    |   movel([0.066867, -1.321516, -2.613726, -0.777146, 1.570796, 1.637663],accel_mss,speed_ms,0,blend_radius_m)
    |   movel([0.067167, -1.321241, -2.613897, -0.777250, 1.570796, 1.637963],accel_mss,speed_ms,0,blend_radius_m)
    |   movel([0.067720, -1.320799, -2.614173, -0.777418, 1.570796, 1.638516],accel_mss,speed_ms,0,blend_radius_m)
    |   movel([0.068900, -1.319924, -2.614716, -0.777749, 1.570796, 1.639696],accel_mss,speed_ms,0,blend_radius_m)
    |   movel([0.070231, -1.318957, -2.615316, -0.778116, 1.570796, 1.641027],accel_mss,speed_ms,0,blend_radius_m)
    |   movel([0.071504, -1.318055, -2.615874, -0.778460, 1.570796, 1.642300],accel_mss,speed_ms,0,blend_radius_m)
    |   movel([0.073287, -1.316906, -2.616583, -0.778900, 1.570796, 1.644084],accel_mss,speed_ms,0,blend_radius_m)
    |   movel([0.076248, -1.315195, -2.617636, -0.779558, 1.570796, 1.647044],accel_mss,speed_ms,0,blend_radius_m)
    |   movel([0.079336, -1.313494, -2.618679, -0.780215, 1.570796, 1.650133],accel_mss,speed_ms,0,blend_radius_m)
    |   movel([0.081717, -1.312291, -2.619415, -0.780683, 1.570796, 1.652514],accel_mss,speed_ms,0,blend_radius_m)
    |   movel([0.083889, -1.311300, -2.620019, -0.781070, 1.570796, 1.654686],accel_mss,speed_ms,0,blend_radius_m)
    |   movel([0.085940, -1.310444, -2.620540, -0.781405, 1.570796, 1.656736],accel_mss,speed_ms,0,blend_radius_m)
    |   movel([0.088113, -1.309632, -2.621034, -0.781723, 1.570796, 1.658909],accel_mss,speed_ms,0,blend_radius_m)
    |   movel([0.090652, -1.308770, -2.621556, -0.782062, 1.570796, 1.661449],accel_mss,speed_ms,0,blend_radius_m)
    |   movel([0.093223, -1.307968, -2.622042, -0.782379, 1.570796, 1.664019],accel_mss,speed_ms,0,blend_radius_m)
    |   movel([0.095145, -1.307454, -2.622353, -0.782582, 1.570796, 1.665941],accel_mss,speed_ms,0,blend_radius_m)
    |   movel([0.096536, -1.307182, -2.622517, -0.782690, 1.570796, 1.667333],accel_mss,speed_ms,0,blend_radius_m)
    |   movel([0.097274, -1.307208, -2.622501, -0.782680, 1.570796, 1.668070],accel_mss,speed_ms,0,blend_radius_m)
    |   movel([0.097500, -1.307382, -2.622396, -0.782611, 1.570796, 1.668297],accel_mss,speed_ms,0,blend_radius_m)
    |   movel([0.097411, -1.307944, -2.622056, -0.782389, 1.570796, 1.668208],accel_mss,speed_ms,0,blend_radius_m)
    |   movel([0.097336, -1.308222, -2.621888, -0.782279, 1.570796, 1.668132],accel_mss,speed_ms,0,blend_radius_m)
    |   movel([0.097240, -1.308511, -2.621713, -0.782165, 1.570796, 1.668037],accel_mss,speed_ms,0,blend_radius_m)
    |   movel([0.097140, -1.308774, -2.621554, -0.782061, 1.570796, 1.667936],accel_mss,speed_ms,0,blend_radius_m)
    |   speed_ms = 0.003
    |   movel([0.097054, -1.295189, -2.614952, -0.802248, 1.570796, 1.667851],accel_mss,speed_ms,0,blend_radius_m)
    |   speed_ms = 1.000
    |   movel([0.097054, -1.268961, -2.601575, -0.841853, 1.570796, 1.667851],accel_mss,speed_ms,0,blend_radius_m)
    |   movel([0.095455, -1.266877, -2.602766, -0.842746, 1.570796, 1.666251],accel_mss,speed_ms,0,blend_radius_m)
    |   movel([0.095455, -1.293135, -2.616170, -0.803084, 1.570796, 1.666251],accel_mss,speed_ms,0,blend_radius_m)
    |   speed_ms = 0.003
    |   movel([0.095455, -1.303429, -2.621063, -0.787897, 1.570796, 1.666251],accel_mss,speed_ms,0,blend_radius_m)
    |   speed_ms = 0.007
    |   movel([0.094815, -1.303693, -2.620905, -0.787791, 1.570796, 1.665611],accel_mss,speed_ms,0,blend_radius_m)
    |   movel([0.093768, -1.303954, -2.620748, -0.787687, 1.570796, 1.664565],accel_mss,speed_ms,0,blend_radius_m)
    |   movel([0.093133, -1.304102, -2.620659, -0.787628, 1.570796, 1.663930],accel_mss,speed_ms,0,blend_radius_m)
    |   movel([0.092577, -1.304211, -2.620593, -0.787584, 1.570796, 1.663373],accel_mss,speed_ms,0,blend_radius_m)
    |   movel([0.092119, -1.304286, -2.620548, -0.787555, 1.570796, 1.662915],accel_mss,speed_ms,0,blend_radius_m)
    |   movel([0.091857, -1.304106, -2.620657, -0.787627, 1.570796, 1.662654],accel_mss,speed_ms,0,blend_radius_m)
    |   movel([0.091804, -1.303854, -2.620808, -0.787727, 1.570796, 1.662600],accel_mss,speed_ms,0,blend_radius_m)
    |   movel([0.091848, -1.303588, -2.620968, -0.787833, 1.570796, 1.662644],accel_mss,speed_ms,0,blend_radius_m)
    |   movel([0.092415, -1.303110, -2.621254, -0.788024, 1.570796, 1.663211],accel_mss,speed_ms,0,blend_radius_m)
    |   movel([0.093796, -1.302701, -2.621500, -0.788188, 1.570796, 1.664592],accel_mss,speed_ms,0,blend_radius_m)
    |   movel([0.095147, -1.302357, -2.621706, -0.788326, 1.570796, 1.665943],accel_mss,speed_ms,0,blend_radius_m)
    |   movel([0.095680, -1.302353, -2.621709, -0.788328, 1.570796, 1.666476],accel_mss,speed_ms,0,blend_radius_m)
    |   movel([0.095880, -1.302466, -2.621641, -0.788282, 1.570796, 1.666676],accel_mss,speed_ms,0,blend_radius_m)
    |   movel([0.095874, -1.302908, -2.621376, -0.788105, 1.570796, 1.666670],accel_mss,speed_ms,0,blend_radius_m)
    |   movel([0.095665, -1.303223, -2.621187, -0.787979, 1.570796, 1.666461],accel_mss,speed_ms,0,blend_radius_m)
    |   speed_ms = 0.003
    |   movel([0.095455, -1.306916, -2.622678, -0.782796, 1.570796, 1.666251],accel_mss,speed_ms,0,blend_radius_m)
    |   speed_ms = 0.007
    |   movel([0.094815, -1.307179, -2.622519, -0.782691, 1.570796, 1.665611],accel_mss,speed_ms,0,blend_radius_m)
    |   movel([0.093768, -1.307439, -2.622362, -0.782588, 1.570796, 1.664565],accel_mss,speed_ms,0,blend_radius_m)
    |   movel([0.093133, -1.307587, -2.622272, -0.782530, 1.570796, 1.663930],accel_mss,speed_ms,0,blend_radius_m)
    |   movel([0.092577, -1.307696, -2.622206, -0.782487, 1.570796, 1.663373],accel_mss,speed_ms,0,blend_radius_m)
    |   movel([0.092119, -1.307771, -2.622161, -0.782457, 1.570796, 1.662915],accel_mss,speed_ms,0,blend_radius_m)
    |   movel([0.091857, -1.307590, -2.622270, -0.782528, 1.570796, 1.662654],accel_mss,speed_ms,0,blend_radius_m)
    |   movel([0.091804, -1.307340, -2.622422, -0.782628, 1.570796, 1.662600],accel_mss,speed_ms,0,blend_radius_m)
    |   movel([0.091848, -1.307074, -2.622582, -0.782733, 1.570796, 1.662644],accel_mss,speed_ms,0,blend_radius_m)
    |   movel([0.092415, -1.306598, -2.622870, -0.782922, 1.570796, 1.663211],accel_mss,speed_ms,0,blend_radius_m)
    |   movel([0.093796, -1.306189, -2.623116, -0.783084, 1.570796, 1.664592],accel_mss,speed_ms,0,blend_radius_m)
    |   movel([0.095147, -1.305846, -2.623322, -0.783220, 1.570796, 1.665943],accel_mss,speed_ms,0,blend_radius_m)
    |   movel([0.095680, -1.305842, -2.623325, -0.783222, 1.570796, 1.666476],accel_mss,speed_ms,0,blend_radius_m)
    |   movel([0.095880, -1.305954, -2.623257, -0.783177, 1.570796, 1.666676],accel_mss,speed_ms,0,blend_radius_m)
    |   movel([0.095874, -1.306395, -2.622992, -0.783002, 1.570796, 1.666670],accel_mss,speed_ms,0,blend_radius_m)
    |   movel([0.095665, -1.306710, -2.622802, -0.782877, 1.570796, 1.666461],accel_mss,speed_ms,0,blend_radius_m)
    |   speed_ms = 0.003
    |   movel([0.095455, -1.293135, -2.616170, -0.803084, 1.570796, 1.666251],accel_mss,speed_ms,0,blend_radius_m)
    |   speed_ms = 1.000
    |   movel([0.095455, -1.266877, -2.602766, -0.842746, 1.570796, 1.666251],accel_mss,speed_ms,0,blend_radius_m)
    |   movel([0.095405, -1.265298, -2.603664, -0.843426, 1.570796, 1.666201],accel_mss,speed_ms,0,blend_radius_m)
    |   movel([0.095405, -1.291578, -2.617089, -0.803722, 1.570796, 1.666201],accel_mss,speed_ms,0,blend_radius_m)
    |   speed_ms = 0.003
    |   movel([0.095405, -1.301882, -2.621990, -0.788516, 1.570796, 1.666201],accel_mss,speed_ms,0,blend_radius_m)
    |   speed_ms = 0.007
    |   movel([0.093973, -1.302304, -2.621738, -0.788347, 1.570796, 1.664770],accel_mss,speed_ms,0,blend_radius_m)
    |   movel([0.092537, -1.302698, -2.621502, -0.788189, 1.570796, 1.663334],accel_mss,speed_ms,0,blend_radius_m)
    |   movel([0.092269, -1.302658, -2.621526, -0.788205, 1.570796, 1.663065],accel_mss,speed_ms,0,blend_radius_m)
    |   movel([0.092184, -1.302449, -2.621651, -0.788289, 1.570796, 1.662981],accel_mss,speed_ms,0,blend_radius_m)
    |   movel([0.092128, -1.302079, -2.621873, -0.788437, 1.570796, 1.662924],accel_mss,speed_ms,0,blend_radius_m)
    |   movel([0.092124, -1.301814, -2.622031, -0.788544, 1.570796, 1.662920],accel_mss,speed_ms,0,blend_radius_m)
    |   movel([0.092244, -1.301453, -2.622247, -0.788689, 1.570796, 1.663040],accel_mss,speed_ms,0,blend_radius_m)
    |   movel([0.093053, -1.300803, -2.622635, -0.788951, 1.570796, 1.663849],accel_mss,speed_ms,0,blend_radius_m)
    |   movel([0.094199, -1.300463, -2.622838, -0.789088, 1.570796, 1.664996],accel_mss,speed_ms,0,blend_radius_m)
    |   movel([0.095309, -1.300319, -2.622924, -0.789146, 1.570796, 1.666105],accel_mss,speed_ms,0,blend_radius_m)
    |   movel([0.095864, -1.300514, -2.622808, -0.789067, 1.570796, 1.666660],accel_mss,speed_ms,0,blend_radius_m)
    |   movel([0.095977, -1.300744, -2.622670, -0.788974, 1.570796, 1.666773],accel_mss,speed_ms,0,blend_radius_m)
    |   movel([0.095993, -1.301082, -2.622469, -0.788838, 1.570796, 1.666789],accel_mss,speed_ms,0,blend_radius_m)
    |   movel([0.095919, -1.301425, -2.622264, -0.788700, 1.570796, 1.666715],accel_mss,speed_ms,0,blend_radius_m)
    |   movel([0.095405, -1.301882, -2.621990, -0.788516, 1.570796, 1.666201],accel_mss,speed_ms,0,blend_radius_m)
    |   speed_ms = 0.003
    |   movel([0.095405, -1.305372, -2.623608, -0.783409, 1.570796, 1.666201],accel_mss,speed_ms,0,blend_radius_m)
    |   speed_ms = 0.007
    |   movel([0.093973, -1.305793, -2.623354, -0.783242, 1.570796, 1.664770],accel_mss,speed_ms,0,blend_radius_m)
    |   movel([0.092537, -1.306187, -2.623117, -0.783085, 1.570796, 1.663334],accel_mss,speed_ms,0,blend_radius_m)
    |   movel([0.092269, -1.306146, -2.623142, -0.783101, 1.570796, 1.663065],accel_mss,speed_ms,0,blend_radius_m)
    |   movel([0.092184, -1.305938, -2.623267, -0.783184, 1.570796, 1.662981],accel_mss,speed_ms,0,blend_radius_m)
    |   movel([0.092128, -1.305569, -2.623489, -0.783331, 1.570796, 1.662924],accel_mss,speed_ms,0,blend_radius_m)
    |   movel([0.092124, -1.305304, -2.623649, -0.783437, 1.570796, 1.662920],accel_mss,speed_ms,0,blend_radius_m)
    |   movel([0.092244, -1.304944, -2.623865, -0.783580, 1.570796, 1.663040],accel_mss,speed_ms,0,blend_radius_m)
    |   movel([0.093053, -1.304296, -2.624254, -0.783839, 1.570796, 1.663849],accel_mss,speed_ms,0,blend_radius_m)
    |   movel([0.094199, -1.303956, -2.624458, -0.783975, 1.570796, 1.664996],accel_mss,speed_ms,0,blend_radius_m)
    |   movel([0.095309, -1.303812, -2.624544, -0.784033, 1.570796, 1.666105],accel_mss,speed_ms,0,blend_radius_m)
    |   movel([0.095864, -1.304007, -2.624428, -0.783955, 1.570796, 1.666660],accel_mss,speed_ms,0,blend_radius_m)
    |   movel([0.095977, -1.304237, -2.624289, -0.783863, 1.570796, 1.666773],accel_mss,speed_ms,0,blend_radius_m)
    |   movel([0.095993, -1.304573, -2.624088, -0.783728, 1.570796, 1.666789],accel_mss,speed_ms,0,blend_radius_m)
    |   movel([0.095919, -1.304916, -2.623882, -0.783591, 1.570796, 1.666715],accel_mss,speed_ms,0,blend_radius_m)
    |   movel([0.095405, -1.305372, -2.623608, -0.783409, 1.570796, 1.666201],accel_mss,speed_ms,0,blend_radius_m)
    |   speed_ms = 0.003
    |   movel([0.095405, -1.291578, -2.617089, -0.803722, 1.570796, 1.666201],accel_mss,speed_ms,0,blend_radius_m)
    |   speed_ms = 1.000
    |   movel([0.095405, -1.265298, -2.603664, -0.843426, 1.570796, 1.666201],accel_mss,speed_ms,0,blend_radius_m)
    |   movel([0.086620, -1.269064, -2.601516, -0.841809, 1.570796, 1.657416],accel_mss,speed_ms,0,blend_radius_m)
    |   movel([0.086620, -1.295291, -2.614891, -0.802207, 1.570796, 1.657416],accel_mss,speed_ms,0,blend_radius_m)
    |   speed_ms = 0.003
    |   movel([0.086620, -1.305571, -2.619774, -0.787044, 1.570796, 1.657416],accel_mss,speed_ms,0,blend_radius_m)
    |   speed_ms = 0.007
    |   movel([0.086582, -1.306010, -2.619509, -0.786870, 1.570796, 1.657378],accel_mss,speed_ms,0,blend_radius_m)
    |   movel([0.086379, -1.306296, -2.619337, -0.786757, 1.570796, 1.657175],accel_mss,speed_ms,0,blend_radius_m)
    |   movel([0.085833, -1.306567, -2.619173, -0.786649, 1.570796, 1.656630],accel_mss,speed_ms,0,blend_radius_m)
    |   movel([0.085166, -1.306876, -2.618986, -0.786527, 1.570796, 1.655962],accel_mss,speed_ms,0,blend_radius_m)
    |   movel([0.084376, -1.307221, -2.618777, -0.786391, 1.570796, 1.655172],accel_mss,speed_ms,0,blend_radius_m)
    |   movel([0.082276, -1.308128, -2.618228, -0.786033, 1.570796, 1.653073],accel_mss,speed_ms,0,blend_radius_m)
    |   movel([0.080804, -1.308806, -2.617816, -0.785767, 1.570796, 1.651600],accel_mss,speed_ms,0,blend_radius_m)
    |   movel([0.079595, -1.309416, -2.617445, -0.785528, 1.570796, 1.650391],accel_mss,speed_ms,0,blend_radius_m)
    |   movel([0.078387, -1.310089, -2.617036, -0.785264, 1.570796, 1.649183],accel_mss,speed_ms,0,blend_radius_m)
    |   movel([0.077797, -1.310425, -2.616831, -0.785133, 1.570796, 1.648593],accel_mss,speed_ms,0,blend_radius_m)
    |   movel([0.077272, -1.310708, -2.616659, -0.785023, 1.570796, 1.648069],accel_mss,speed_ms,0,blend_radius_m)
    |   movel([0.076832, -1.310931, -2.616522, -0.784935, 1.570796, 1.647629],accel_mss,speed_ms,0,blend_radius_m)
    |   movel([0.076556, -1.310865, -2.616563, -0.784961, 1.570796, 1.647352],accel_mss,speed_ms,0,blend_radius_m)
    |   movel([0.076460, -1.310625, -2.616709, -0.785055, 1.570796, 1.647257],accel_mss,speed_ms,0,blend_radius_m)
    |   movel([0.076484, -1.310298, -2.616908, -0.785183, 1.570796, 1.647280],accel_mss,speed_ms,0,blend_radius_m)
    |   movel([0.076654, -1.309989, -2.617097, -0.785303, 1.570796, 1.647450],accel_mss,speed_ms,0,blend_radius_m)
    |   movel([0.077020, -1.309644, -2.617307, -0.785438, 1.570796, 1.647816],accel_mss,speed_ms,0,blend_radius_m)
    |   movel([0.077663, -1.309194, -2.617580, -0.785615, 1.570796, 1.648459],accel_mss,speed_ms,0,blend_radius_m)
    |   movel([0.078607, -1.308648, -2.617912, -0.785829, 1.570796, 1.649403],accel_mss,speed_ms,0,blend_radius_m)
    |   movel([0.080873, -1.307513, -2.618601, -0.786276, 1.570796, 1.651669],accel_mss,speed_ms,0,blend_radius_m)
    |   movel([0.083162, -1.306405, -2.619271, -0.786713, 1.570796, 1.653958],accel_mss,speed_ms,0,blend_radius_m)
    |   movel([0.084650, -1.305747, -2.619668, -0.786974, 1.570796, 1.655447],accel_mss,speed_ms,0,blend_radius_m)
    |   movel([0.085312, -1.305509, -2.619812, -0.787068, 1.570796, 1.656108],accel_mss,speed_ms,0,blend_radius_m)
    |   movel([0.085892, -1.305370, -2.619896, -0.787124, 1.570796, 1.656689],accel_mss,speed_ms,0,blend_radius_m)
    |   movel([0.086338, -1.305334, -2.619917, -0.787138, 1.570796, 1.657135],accel_mss,speed_ms,0,blend_radius_m)
    |   movel([0.086557, -1.305429, -2.619860, -0.787100, 1.570796, 1.657353],accel_mss,speed_ms,0,blend_radius_m)
    |   speed_ms = 0.003
    |   movel([0.086620, -1.309053, -2.621385, -0.781951, 1.570796, 1.657416],accel_mss,speed_ms,0,blend_radius_m)
    |   speed_ms = 0.007
    |   movel([0.086582, -1.309490, -2.621120, -0.781779, 1.570796, 1.657378],accel_mss,speed_ms,0,blend_radius_m)
    |   movel([0.086379, -1.309776, -2.620947, -0.781667, 1.570796, 1.657175],accel_mss,speed_ms,0,blend_radius_m)
    |   movel([0.085833, -1.310046, -2.620782, -0.781561, 1.570796, 1.656630],accel_mss,speed_ms,0,blend_radius_m)
    |   movel([0.085166, -1.310354, -2.620595, -0.781440, 1.570796, 1.655962],accel_mss,speed_ms,0,blend_radius_m)
    |   movel([0.084376, -1.310699, -2.620385, -0.781305, 1.570796, 1.655172],accel_mss,speed_ms,0,blend_radius_m)
    |   movel([0.082276, -1.311603, -2.619834, -0.780951, 1.570796, 1.653073],accel_mss,speed_ms,0,blend_radius_m)
    |   movel([0.080804, -1.312280, -2.619421, -0.780687, 1.570796, 1.651600],accel_mss,speed_ms,0,blend_radius_m)
    |   movel([0.079595, -1.312889, -2.619050, -0.780450, 1.570796, 1.650391],accel_mss,speed_ms,0,blend_radius_m)
    |   movel([0.078387, -1.313560, -2.618639, -0.780190, 1.570796, 1.649183],accel_mss,speed_ms,0,blend_radius_m)
    |   movel([0.077797, -1.313896, -2.618434, -0.780060, 1.570796, 1.648593],accel_mss,speed_ms,0,blend_radius_m)
    |   movel([0.077272, -1.314177, -2.618261, -0.779951, 1.570796, 1.648069],accel_mss,speed_ms,0,blend_radius_m)
    |   movel([0.076832, -1.314401, -2.618124, -0.779864, 1.570796, 1.647629],accel_mss,speed_ms,0,blend_radius_m)
    |   movel([0.076556, -1.314335, -2.618165, -0.779890, 1.570796, 1.647352],accel_mss,speed_ms,0,blend_radius_m)
    |   movel([0.076460, -1.314095, -2.618312, -0.779983, 1.570796, 1.647257],accel_mss,speed_ms,0,blend_radius_m)
    |   movel([0.076484, -1.313769, -2.618511, -0.780109, 1.570796, 1.647280],accel_mss,speed_ms,0,blend_radius_m)
    |   movel([0.076654, -1.313460, -2.618700, -0.780229, 1.570796, 1.647450],accel_mss,speed_ms,0,blend_radius_m)
    |   movel([0.077020, -1.313116, -2.618911, -0.780362, 1.570796, 1.647816],accel_mss,speed_ms,0,blend_radius_m)
    |   movel([0.077663, -1.312667, -2.619185, -0.780537, 1.570796, 1.648459],accel_mss,speed_ms,0,blend_radius_m)
    |   movel([0.078607, -1.312122, -2.619518, -0.780749, 1.570796, 1.649403],accel_mss,speed_ms,0,blend_radius_m)
    |   movel([0.080873, -1.310990, -2.620208, -0.781191, 1.570796, 1.651669],accel_mss,speed_ms,0,blend_radius_m)
    |   movel([0.083162, -1.309885, -2.620880, -0.781624, 1.570796, 1.653958],accel_mss,speed_ms,0,blend_radius_m)
    |   movel([0.084650, -1.309228, -2.621279, -0.781882, 1.570796, 1.655447],accel_mss,speed_ms,0,blend_radius_m)
    |   movel([0.085312, -1.308990, -2.621423, -0.781976, 1.570796, 1.656108],accel_mss,speed_ms,0,blend_radius_m)
    |   movel([0.085892, -1.308852, -2.621507, -0.782030, 1.570796, 1.656689],accel_mss,speed_ms,0,blend_radius_m)
    |   movel([0.086338, -1.308816, -2.621529, -0.782044, 1.570796, 1.657135],accel_mss,speed_ms,0,blend_radius_m)
    |   movel([0.086557, -1.308911, -2.621471, -0.782007, 1.570796, 1.657353],accel_mss,speed_ms,0,blend_radius_m)
    |   speed_ms = 0.003
    |   movel([0.086620, -1.295291, -2.614891, -0.802207, 1.570796, 1.657416],accel_mss,speed_ms,0,blend_radius_m)
    |   speed_ms = 1.000
    |   movel([0.086620, -1.269064, -2.601516, -0.841809, 1.570796, 1.657416],accel_mss,speed_ms,0,blend_radius_m)
    |   movel([0.086236, -1.268202, -2.602010, -0.842178, 1.570796, 1.657033],accel_mss,speed_ms,0,blend_radius_m)
    |   movel([0.086236, -1.294441, -2.615396, -0.802552, 1.570796, 1.657033],accel_mss,speed_ms,0,blend_radius_m)
    |   speed_ms = 0.003
    |   movel([0.086236, -1.304727, -2.620283, -0.787379, 1.570796, 1.657033],accel_mss,speed_ms,0,blend_radius_m)
    |   speed_ms = 0.007
    |   movel([0.085836, -1.304918, -2.620168, -0.787303, 1.570796, 1.656632],accel_mss,speed_ms,0,blend_radius_m)
    |   movel([0.085399, -1.305046, -2.620090, -0.787252, 1.570796, 1.656196],accel_mss,speed_ms,0,blend_radius_m)
    |   movel([0.085110, -1.304940, -2.620155, -0.787294, 1.570796, 1.655906],accel_mss,speed_ms,0,blend_radius_m)
    |   movel([0.085056, -1.304704, -2.620297, -0.787388, 1.570796, 1.655852],accel_mss,speed_ms,0,blend_radius_m)
    |   movel([0.085010, -1.304411, -2.620473, -0.787505, 1.570796, 1.655807],accel_mss,speed_ms,0,blend_radius_m)
    |   movel([0.084978, -1.304084, -2.620670, -0.787635, 1.570796, 1.655775],accel_mss,speed_ms,0,blend_radius_m)
    |   movel([0.084892, -1.303468, -2.621040, -0.787881, 1.570796, 1.655688],accel_mss,speed_ms,0,blend_radius_m)
    |   movel([0.084735, -1.303084, -2.621270, -0.788035, 1.570796, 1.655531],accel_mss,speed_ms,0,blend_radius_m)
    |   movel([0.084474, -1.302865, -2.621402, -0.788122, 1.570796, 1.655271],accel_mss,speed_ms,0,blend_radius_m)
    |   movel([0.084085, -1.302763, -2.621463, -0.788163, 1.570796, 1.654882],accel_mss,speed_ms,0,blend_radius_m)
    |   movel([0.083756, -1.302782, -2.621451, -0.788155, 1.570796, 1.654553],accel_mss,speed_ms,0,blend_radius_m)
    |   movel([0.083385, -1.302888, -2.621388, -0.788113, 1.570796, 1.654181],accel_mss,speed_ms,0,blend_radius_m)
    |   movel([0.082789, -1.303141, -2.621236, -0.788012, 1.570796, 1.653585],accel_mss,speed_ms,0,blend_radius_m)
    |   movel([0.081437, -1.303782, -2.620851, -0.787756, 1.570796, 1.652233],accel_mss,speed_ms,0,blend_radius_m)
    |   movel([0.079639, -1.304655, -2.620326, -0.787408, 1.570796, 1.650435],accel_mss,speed_ms,0,blend_radius_m)
    |   movel([0.078834, -1.305092, -2.620063, -0.787234, 1.570796, 1.649630],accel_mss,speed_ms,0,blend_radius_m)
    |   movel([0.078346, -1.305441, -2.619853, -0.787095, 1.570796, 1.649142],accel_mss,speed_ms,0,blend_radius_m)
    |   movel([0.077948, -1.305852, -2.619605, -0.786932, 1.570796, 1.648744],accel_mss,speed_ms,0,blend_radius_m)
    |   movel([0.077690, -1.306269, -2.619353, -0.786767, 1.570796, 1.648486],accel_mss,speed_ms,0,blend_radius_m)
    |   movel([0.077544, -1.306721, -2.619080, -0.786588, 1.570796, 1.648340],accel_mss,speed_ms,0,blend_radius_m)
    |   movel([0.077508, -1.307216, -2.618780, -0.786393, 1.570796, 1.648304],accel_mss,speed_ms,0,blend_radius_m)
    |   movel([0.077587, -1.307758, -2.618452, -0.786179, 1.570796, 1.648383],accel_mss,speed_ms,0,blend_radius_m)
    |   movel([0.077671, -1.308128, -2.618228, -0.786033, 1.570796, 1.648467],accel_mss,speed_ms,0,blend_radius_m)
    |   movel([0.077735, -1.308415, -2.618054, -0.785921, 1.570796, 1.648531],accel_mss,speed_ms,0,blend_radius_m)
    |   movel([0.077659, -1.308677, -2.617895, -0.785818, 1.570796, 1.648455],accel_mss,speed_ms,0,blend_radius_m)
    |   movel([0.077187, -1.309039, -2.617674, -0.785675, 1.570796, 1.647984],accel_mss,speed_ms,0,blend_radius_m)
    |   movel([0.076724, -1.309309, -2.617511, -0.785570, 1.570796, 1.647520],accel_mss,speed_ms,0,blend_radius_m)
    |   movel([0.076338, -1.309187, -2.617585, -0.785618, 1.570796, 1.647134],accel_mss,speed_ms,0,blend_radius_m)
    |   movel([0.076209, -1.308628, -2.617924, -0.785837, 1.570796, 1.647005],accel_mss,speed_ms,0,blend_radius_m)
    |   movel([0.076116, -1.307960, -2.618330, -0.786100, 1.570796, 1.646913],accel_mss,speed_ms,0,blend_radius_m)
    |   movel([0.076083, -1.307280, -2.618742, -0.786368, 1.570796, 1.646879],accel_mss,speed_ms,0,blend_radius_m)
    |   movel([0.076095, -1.306774, -2.619048, -0.786567, 1.570796, 1.646891],accel_mss,speed_ms,0,blend_radius_m)
    |   movel([0.076142, -1.306449, -2.619244, -0.786696, 1.570796, 1.646938],accel_mss,speed_ms,0,blend_radius_m)
    |   movel([0.076248, -1.306149, -2.619426, -0.786815, 1.570796, 1.647044],accel_mss,speed_ms,0,blend_radius_m)
    |   movel([0.076446, -1.305763, -2.619659, -0.786968, 1.570796, 1.647243],accel_mss,speed_ms,0,blend_radius_m)
    |   movel([0.076797, -1.305253, -2.619966, -0.787170, 1.570796, 1.647593],accel_mss,speed_ms,0,blend_radius_m)
    |   movel([0.077222, -1.304834, -2.620218, -0.787337, 1.570796, 1.648018],accel_mss,speed_ms,0,blend_radius_m)
    |   movel([0.077828, -1.304417, -2.620470, -0.787503, 1.570796, 1.648625],accel_mss,speed_ms,0,blend_radius_m)
    |   movel([0.078794, -1.303880, -2.620792, -0.787717, 1.570796, 1.649591],accel_mss,speed_ms,0,blend_radius_m)
    |   movel([0.080203, -1.303163, -2.621223, -0.788003, 1.570796, 1.651000],accel_mss,speed_ms,0,blend_radius_m)
    |   movel([0.081785, -1.302416, -2.621671, -0.788302, 1.570796, 1.652581],accel_mss,speed_ms,0,blend_radius_m)
    |   movel([0.083247, -1.301763, -2.622062, -0.788564, 1.570796, 1.654043],accel_mss,speed_ms,0,blend_radius_m)
    |   movel([0.084162, -1.301411, -2.622272, -0.788706, 1.570796, 1.654958],accel_mss,speed_ms,0,blend_radius_m)
    |   movel([0.084675, -1.301251, -2.622368, -0.788770, 1.570796, 1.655472],accel_mss,speed_ms,0,blend_radius_m)
    |   movel([0.084988, -1.301189, -2.622405, -0.788795, 1.570796, 1.655784],accel_mss,speed_ms,0,blend_radius_m)
    |   movel([0.085477, -1.301278, -2.622352, -0.788759, 1.570796, 1.656273],accel_mss,speed_ms,0,blend_radius_m)
    |   movel([0.085801, -1.301477, -2.622233, -0.788679, 1.570796, 1.656597],accel_mss,speed_ms,0,blend_radius_m)
    |   movel([0.086025, -1.301709, -2.622094, -0.788586, 1.570796, 1.656822],accel_mss,speed_ms,0,blend_radius_m)
    |   movel([0.086213, -1.302208, -2.621795, -0.788386, 1.570796, 1.657010],accel_mss,speed_ms,0,blend_radius_m)
    |   movel([0.086374, -1.303118, -2.621250, -0.788021, 1.570796, 1.657170],accel_mss,speed_ms,0,blend_radius_m)
    |   movel([0.086472, -1.304054, -2.620688, -0.787647, 1.570796, 1.657269],accel_mss,speed_ms,0,blend_radius_m)
    |   movel([0.086421, -1.304572, -2.620376, -0.787441, 1.570796, 1.657218],accel_mss,speed_ms,0,blend_radius_m)
    |   speed_ms = 0.003
    |   movel([0.086236, -1.308210, -2.621895, -0.782283, 1.570796, 1.657033],accel_mss,speed_ms,0,blend_radius_m)
    |   speed_ms = 0.007
    |   movel([0.085836, -1.308401, -2.621780, -0.782208, 1.570796, 1.656632],accel_mss,speed_ms,0,blend_radius_m)
    |   movel([0.085399, -1.308529, -2.621702, -0.782158, 1.570796, 1.656196],accel_mss,speed_ms,0,blend_radius_m)
    |   movel([0.085110, -1.308423, -2.621767, -0.782199, 1.570796, 1.655906],accel_mss,speed_ms,0,blend_radius_m)
    |   movel([0.085056, -1.308187, -2.621909, -0.782292, 1.570796, 1.655852],accel_mss,speed_ms,0,blend_radius_m)
    |   movel([0.085010, -1.307895, -2.622086, -0.782408, 1.570796, 1.655807],accel_mss,speed_ms,0,blend_radius_m)
    |   movel([0.084978, -1.307569, -2.622283, -0.782537, 1.570796, 1.655775],accel_mss,speed_ms,0,blend_radius_m)
    |   movel([0.084892, -1.306955, -2.622654, -0.782780, 1.570796, 1.655688],accel_mss,speed_ms,0,blend_radius_m)
    |   movel([0.084735, -1.306571, -2.622886, -0.782932, 1.570796, 1.655531],accel_mss,speed_ms,0,blend_radius_m)
    |   movel([0.084474, -1.306352, -2.623017, -0.783019, 1.570796, 1.655271],accel_mss,speed_ms,0,blend_radius_m)
    |   movel([0.084085, -1.306251, -2.623078, -0.783059, 1.570796, 1.654882],accel_mss,speed_ms,0,blend_radius_m)
    |   movel([0.083756, -1.306270, -2.623067, -0.783052, 1.570796, 1.654553],accel_mss,speed_ms,0,blend_radius_m)
    |   movel([0.083385, -1.306376, -2.623003, -0.783010, 1.570796, 1.654181],accel_mss,speed_ms,0,blend_radius_m)
    |   movel([0.082789, -1.306629, -2.622851, -0.782910, 1.570796, 1.653585],accel_mss,speed_ms,0,blend_radius_m)
    |   movel([0.081437, -1.307268, -2.622465, -0.782656, 1.570796, 1.652233],accel_mss,speed_ms,0,blend_radius_m)
    |   movel([0.079639, -1.308139, -2.621939, -0.782312, 1.570796, 1.650435],accel_mss,speed_ms,0,blend_radius_m)
    |   movel([0.078834, -1.308575, -2.621675, -0.782140, 1.570796, 1.649630],accel_mss,speed_ms,0,blend_radius_m)
    |   movel([0.078346, -1.308923, -2.621464, -0.782002, 1.570796, 1.649142],accel_mss,speed_ms,0,blend_radius_m)
    |   movel([0.077948, -1.309333, -2.621215, -0.781841, 1.570796, 1.648744],accel_mss,speed_ms,0,blend_radius_m)
    |   movel([0.077690, -1.309749, -2.620962, -0.781677, 1.570796, 1.648486],accel_mss,speed_ms,0,blend_radius_m)
    |   movel([0.077544, -1.310200, -2.620689, -0.781500, 1.570796, 1.648340],accel_mss,speed_ms,0,blend_radius_m)
    |   movel([0.077508, -1.310694, -2.620388, -0.781307, 1.570796, 1.648304],accel_mss,speed_ms,0,blend_radius_m)
    |   movel([0.077587, -1.311234, -2.620059, -0.781095, 1.570796, 1.648383],accel_mss,speed_ms,0,blend_radius_m)
    |   movel([0.077671, -1.311604, -2.619834, -0.780951, 1.570796, 1.648467],accel_mss,speed_ms,0,blend_radius_m)
    |   movel([0.077735, -1.311890, -2.619660, -0.780839, 1.570796, 1.648531],accel_mss,speed_ms,0,blend_radius_m)
    |   movel([0.077659, -1.312151, -2.619500, -0.780738, 1.570796, 1.648455],accel_mss,speed_ms,0,blend_radius_m)
    |   movel([0.077187, -1.312513, -2.619280, -0.780597, 1.570796, 1.647984],accel_mss,speed_ms,0,blend_radius_m)
    |   movel([0.076724, -1.312781, -2.619115, -0.780492, 1.570796, 1.647520],accel_mss,speed_ms,0,blend_radius_m)
    |   movel([0.076338, -1.312660, -2.619190, -0.780540, 1.570796, 1.647134],accel_mss,speed_ms,0,blend_radius_m)
    |   movel([0.076209, -1.312103, -2.619530, -0.780756, 1.570796, 1.647005],accel_mss,speed_ms,0,blend_radius_m)
    |   movel([0.076116, -1.311436, -2.619937, -0.781017, 1.570796, 1.646913],accel_mss,speed_ms,0,blend_radius_m)
    |   movel([0.076083, -1.310757, -2.620350, -0.781282, 1.570796, 1.646879],accel_mss,speed_ms,0,blend_radius_m)
    |   movel([0.076095, -1.310253, -2.620656, -0.781480, 1.570796, 1.646891],accel_mss,speed_ms,0,blend_radius_m)
    |   movel([0.076142, -1.309929, -2.620853, -0.781607, 1.570796, 1.646938],accel_mss,speed_ms,0,blend_radius_m)
    |   movel([0.076248, -1.309629, -2.621036, -0.781725, 1.570796, 1.647044],accel_mss,speed_ms,0,blend_radius_m)
    |   movel([0.076446, -1.309244, -2.621269, -0.781876, 1.570796, 1.647243],accel_mss,speed_ms,0,blend_radius_m)
    |   movel([0.076797, -1.308735, -2.621577, -0.782076, 1.570796, 1.647593],accel_mss,speed_ms,0,blend_radius_m)
    |   movel([0.077222, -1.308317, -2.621831, -0.782241, 1.570796, 1.648018],accel_mss,speed_ms,0,blend_radius_m)
    |   movel([0.077828, -1.307901, -2.622083, -0.782406, 1.570796, 1.648625],accel_mss,speed_ms,0,blend_radius_m)
    |   movel([0.078794, -1.307365, -2.622406, -0.782618, 1.570796, 1.649591],accel_mss,speed_ms,0,blend_radius_m)
    |   movel([0.080203, -1.306650, -2.622838, -0.782901, 1.570796, 1.651000],accel_mss,speed_ms,0,blend_radius_m)
    |   movel([0.081785, -1.305904, -2.623287, -0.783197, 1.570796, 1.652581],accel_mss,speed_ms,0,blend_radius_m)
    |   movel([0.083247, -1.305253, -2.623679, -0.783457, 1.570796, 1.654043],accel_mss,speed_ms,0,blend_radius_m)
    |   movel([0.084162, -1.304902, -2.623890, -0.783597, 1.570796, 1.654958],accel_mss,speed_ms,0,blend_radius_m)
    |   movel([0.084675, -1.304742, -2.623986, -0.783660, 1.570796, 1.655472],accel_mss,speed_ms,0,blend_radius_m)
    |   movel([0.084988, -1.304680, -2.624023, -0.783685, 1.570796, 1.655784],accel_mss,speed_ms,0,blend_radius_m)
    |   movel([0.085477, -1.304770, -2.623970, -0.783650, 1.570796, 1.656273],accel_mss,speed_ms,0,blend_radius_m)
    |   movel([0.085801, -1.304968, -2.623851, -0.783571, 1.570796, 1.656597],accel_mss,speed_ms,0,blend_radius_m)
    |   movel([0.086025, -1.305199, -2.623712, -0.783478, 1.570796, 1.656822],accel_mss,speed_ms,0,blend_radius_m)
    |   movel([0.086213, -1.305697, -2.623412, -0.783280, 1.570796, 1.657010],accel_mss,speed_ms,0,blend_radius_m)
    |   movel([0.086374, -1.306605, -2.622865, -0.782919, 1.570796, 1.657170],accel_mss,speed_ms,0,blend_radius_m)
    |   movel([0.086472, -1.307539, -2.622301, -0.782549, 1.570796, 1.657269],accel_mss,speed_ms,0,blend_radius_m)
    |   movel([0.086421, -1.308056, -2.621989, -0.782344, 1.570796, 1.657218],accel_mss,speed_ms,0,blend_radius_m)
    |   speed_ms = 0.003
    |   movel([0.086236, -1.294441, -2.615396, -0.802552, 1.570796, 1.657033],accel_mss,speed_ms,0,blend_radius_m)
    |   speed_ms = 1.000
    |   movel([0.086236, -1.268202, -2.602010, -0.842178, 1.570796, 1.657033],accel_mss,speed_ms,0,blend_radius_m)
    |   movel([0.090839, -1.274742, -2.598244, -0.839403, 1.570796, 1.661635],accel_mss,speed_ms,0,blend_radius_m)
    |   movel([0.090839, -1.300888, -2.611545, -0.799956, 1.570796, 1.661635],accel_mss,speed_ms,0,blend_radius_m)
    |   speed_ms = 0.003
    |   movel([0.090839, -1.311132, -2.616400, -0.784857, 1.570796, 1.661635],accel_mss,speed_ms,0,blend_radius_m)
    |   speed_ms = 0.007
    |   movel([0.091231, -1.310851, -2.616572, -0.784967, 1.570796, 1.662027],accel_mss,speed_ms,0,blend_radius_m)
    |   movel([0.093076, -1.310222, -2.616955, -0.785212, 1.570796, 1.663872],accel_mss,speed_ms,0,blend_radius_m)
    |   movel([0.094912, -1.309640, -2.617309, -0.785440, 1.570796, 1.665708],accel_mss,speed_ms,0,blend_radius_m)
    |   movel([0.095311, -1.309662, -2.617295, -0.785431, 1.570796, 1.666108],accel_mss,speed_ms,0,blend_radius_m)
    |   movel([0.095304, -1.309901, -2.617150, -0.785338, 1.570796, 1.666100],accel_mss,speed_ms,0,blend_radius_m)
    |   movel([0.094896, -1.310250, -2.616938, -0.785201, 1.570796, 1.665692],accel_mss,speed_ms,0,blend_radius_m)
    |   movel([0.094536, -1.310423, -2.616832, -0.785134, 1.570796, 1.665332],accel_mss,speed_ms,0,blend_radius_m)
    |   movel([0.093961, -1.310638, -2.616701, -0.785050, 1.570796, 1.664758],accel_mss,speed_ms,0,blend_radius_m)
    |   movel([0.092892, -1.310989, -2.616487, -0.784913, 1.570796, 1.663688],accel_mss,speed_ms,0,blend_radius_m)
    |   movel([0.091876, -1.311310, -2.616291, -0.784788, 1.570796, 1.662673],accel_mss,speed_ms,0,blend_radius_m)
    |   movel([0.091309, -1.311465, -2.616196, -0.784727, 1.570796, 1.662105],accel_mss,speed_ms,0,blend_radius_m)
    |   movel([0.090961, -1.311529, -2.616157, -0.784703, 1.570796, 1.661757],accel_mss,speed_ms,0,blend_radius_m)
    |   movel([0.090736, -1.311417, -2.616225, -0.784746, 1.570796, 1.661532],accel_mss,speed_ms,0,blend_radius_m)
    |   movel([0.090839, -1.311132, -2.616400, -0.784857, 1.570796, 1.661635],accel_mss,speed_ms,0,blend_radius_m)
    |   speed_ms = 0.003
    |   movel([0.090839, -1.314601, -2.618001, -0.779787, 1.570796, 1.661635],accel_mss,speed_ms,0,blend_radius_m)
    |   speed_ms = 0.007
    |   movel([0.091231, -1.314320, -2.618174, -0.779896, 1.570796, 1.662027],accel_mss,speed_ms,0,blend_radius_m)
    |   movel([0.093076, -1.313693, -2.618558, -0.780138, 1.570796, 1.663872],accel_mss,speed_ms,0,blend_radius_m)
    |   movel([0.094912, -1.313112, -2.618913, -0.780364, 1.570796, 1.665708],accel_mss,speed_ms,0,blend_radius_m)
    |   movel([0.095311, -1.313135, -2.618899, -0.780355, 1.570796, 1.666108],accel_mss,speed_ms,0,blend_radius_m)
    |   movel([0.095304, -1.313373, -2.618754, -0.780263, 1.570796, 1.666100],accel_mss,speed_ms,0,blend_radius_m)
    |   movel([0.094896, -1.313720, -2.618541, -0.780128, 1.570796, 1.665692],accel_mss,speed_ms,0,blend_radius_m)
    |   movel([0.094536, -1.313893, -2.618435, -0.780061, 1.570796, 1.665332],accel_mss,speed_ms,0,blend_radius_m)
    |   movel([0.093961, -1.314108, -2.618304, -0.779978, 1.570796, 1.664758],accel_mss,speed_ms,0,blend_radius_m)
    |   movel([0.092892, -1.314458, -2.618089, -0.779842, 1.570796, 1.663688],accel_mss,speed_ms,0,blend_radius_m)
    |   movel([0.091876, -1.314778, -2.617893, -0.779719, 1.570796, 1.662673],accel_mss,speed_ms,0,blend_radius_m)
    |   movel([0.091309, -1.314933, -2.617797, -0.779659, 1.570796, 1.662105],accel_mss,speed_ms,0,blend_radius_m)
    |   movel([0.090961, -1.314997, -2.617758, -0.779634, 1.570796, 1.661757],accel_mss,speed_ms,0,blend_radius_m)
    |   movel([0.090736, -1.314885, -2.617826, -0.779677, 1.570796, 1.661532],accel_mss,speed_ms,0,blend_radius_m)
    |   movel([0.090839, -1.314601, -2.618001, -0.779787, 1.570796, 1.661635],accel_mss,speed_ms,0,blend_radius_m)
    |   speed_ms = 0.003
    |   movel([0.090839, -1.300888, -2.611545, -0.799956, 1.570796, 1.661635],accel_mss,speed_ms,0,blend_radius_m)
    |   speed_ms = 1.000
    |   movel([0.090839, -1.274742, -2.598244, -0.839403, 1.570796, 1.661635],accel_mss,speed_ms,0,blend_radius_m)
    |   movel([0.090283, -1.274574, -2.598342, -0.839473, 1.570796, 1.661079],accel_mss,speed_ms,0,blend_radius_m)
    |   movel([0.090283, -1.300723, -2.611644, -0.800022, 1.570796, 1.661079],accel_mss,speed_ms,0,blend_radius_m)
    |   speed_ms = 0.003
    |   movel([0.090283, -1.310968, -2.616500, -0.784921, 1.570796, 1.661079],accel_mss,speed_ms,0,blend_radius_m)
    |   speed_ms = 0.007
    |   movel([0.091304, -1.309341, -2.617491, -0.785557, 1.570796, 1.662100],accel_mss,speed_ms,0,blend_radius_m)
    |   movel([0.091772, -1.308890, -2.617765, -0.785734, 1.570796, 1.662568],accel_mss,speed_ms,0,blend_radius_m)
    |   movel([0.092217, -1.308558, -2.617967, -0.785864, 1.570796, 1.663014],accel_mss,speed_ms,0,blend_radius_m)
    |   movel([0.092713, -1.308300, -2.618123, -0.785966, 1.570796, 1.663510],accel_mss,speed_ms,0,blend_radius_m)
    |   movel([0.093344, -1.308063, -2.618267, -0.786059, 1.570796, 1.664141],accel_mss,speed_ms,0,blend_radius_m)
    |   movel([0.094712, -1.307930, -2.618348, -0.786111, 1.570796, 1.665509],accel_mss,speed_ms,0,blend_radius_m)
    |   movel([0.095678, -1.308467, -2.618022, -0.785900, 1.570796, 1.666474],accel_mss,speed_ms,0,blend_radius_m)
    |   movel([0.096003, -1.309536, -2.617373, -0.785481, 1.570796, 1.666799],accel_mss,speed_ms,0,blend_radius_m)
    |   movel([0.095606, -1.310869, -2.616560, -0.784960, 1.570796, 1.666402],accel_mss,speed_ms,0,blend_radius_m)
    |   movel([0.095281, -1.311375, -2.616251, -0.784763, 1.570796, 1.666077],accel_mss,speed_ms,0,blend_radius_m)
    |   movel([0.094834, -1.311913, -2.615923, -0.784553, 1.570796, 1.665631],accel_mss,speed_ms,0,blend_radius_m)
    |   movel([0.094350, -1.312398, -2.615626, -0.784365, 1.570796, 1.665146],accel_mss,speed_ms,0,blend_radius_m)
    |   movel([0.093908, -1.312733, -2.615421, -0.784235, 1.570796, 1.664704],accel_mss,speed_ms,0,blend_radius_m)
    |   movel([0.093410, -1.312978, -2.615271, -0.784140, 1.570796, 1.664206],accel_mss,speed_ms,0,blend_radius_m)
    |   movel([0.093084, -1.313110, -2.615190, -0.784089, 1.570796, 1.663881],accel_mss,speed_ms,0,blend_radius_m)
    |   movel([0.092771, -1.313220, -2.615122, -0.784047, 1.570796, 1.663568],accel_mss,speed_ms,0,blend_radius_m)
    |   movel([0.091175, -1.313300, -2.615073, -0.784016, 1.570796, 1.661972],accel_mss,speed_ms,0,blend_radius_m)
    |   movel([0.090238, -1.312456, -2.615591, -0.784343, 1.570796, 1.661034],accel_mss,speed_ms,0,blend_radius_m)
    |   movel([0.090283, -1.310968, -2.616500, -0.784921, 1.570796, 1.661079],accel_mss,speed_ms,0,blend_radius_m)
    |   speed_ms = 0.003
    |   movel([0.090283, -1.314437, -2.618102, -0.779850, 1.570796, 1.661079],accel_mss,speed_ms,0,blend_radius_m)
    |   speed_ms = 0.007
    |   movel([0.091304, -1.312814, -2.619095, -0.780479, 1.570796, 1.662100],accel_mss,speed_ms,0,blend_radius_m)
    |   movel([0.091772, -1.312364, -2.619370, -0.780654, 1.570796, 1.662568],accel_mss,speed_ms,0,blend_radius_m)
    |   movel([0.092217, -1.312033, -2.619573, -0.780784, 1.570796, 1.663014],accel_mss,speed_ms,0,blend_radius_m)
    |   movel([0.092713, -1.311775, -2.619730, -0.780884, 1.570796, 1.663510],accel_mss,speed_ms,0,blend_radius_m)
    |   movel([0.093344, -1.311539, -2.619874, -0.780976, 1.570796, 1.664141],accel_mss,speed_ms,0,blend_radius_m)
    |   movel([0.094712, -1.311406, -2.619954, -0.781028, 1.570796, 1.665509],accel_mss,speed_ms,0,blend_radius_m)
    |   movel([0.095678, -1.311942, -2.619628, -0.780819, 1.570796, 1.666474],accel_mss,speed_ms,0,blend_radius_m)
    |   movel([0.096003, -1.313008, -2.618977, -0.780404, 1.570796, 1.666799],accel_mss,speed_ms,0,blend_radius_m)
    |   movel([0.095606, -1.314338, -2.618162, -0.779889, 1.570796, 1.666402],accel_mss,speed_ms,0,blend_radius_m)
    |   movel([0.095281, -1.314843, -2.617852, -0.779693, 1.570796, 1.666077],accel_mss,speed_ms,0,blend_radius_m)
    |   movel([0.094834, -1.315380, -2.617523, -0.779486, 1.570796, 1.665631],accel_mss,speed_ms,0,blend_radius_m)
    |   movel([0.094350, -1.315864, -2.617225, -0.779300, 1.570796, 1.665146],accel_mss,speed_ms,0,blend_radius_m)
    |   movel([0.093908, -1.316198, -2.617019, -0.779171, 1.570796, 1.664704],accel_mss,speed_ms,0,blend_radius_m)
    |   movel([0.093410, -1.316443, -2.616869, -0.779078, 1.570796, 1.664206],accel_mss,speed_ms,0,blend_radius_m)
    |   movel([0.093084, -1.316574, -2.616788, -0.779027, 1.570796, 1.663881],accel_mss,speed_ms,0,blend_radius_m)
    |   movel([0.092771, -1.316684, -2.616720, -0.778985, 1.570796, 1.663568],accel_mss,speed_ms,0,blend_radius_m)
    |   movel([0.091175, -1.316764, -2.616671, -0.778954, 1.570796, 1.661972],accel_mss,speed_ms,0,blend_radius_m)
    |   movel([0.090238, -1.315921, -2.617190, -0.779278, 1.570796, 1.661034],accel_mss,speed_ms,0,blend_radius_m)
    |   movel([0.090283, -1.314437, -2.618102, -0.779850, 1.570796, 1.661079],accel_mss,speed_ms,0,blend_radius_m)
    |   speed_ms = 0.003
    |   movel([0.090283, -1.300723, -2.611644, -0.800022, 1.570796, 1.661079],accel_mss,speed_ms,0,blend_radius_m)
    |   speed_ms = 1.000
    |   movel([0.090283, -1.274574, -2.598342, -0.839473, 1.570796, 1.661079],accel_mss,speed_ms,0,blend_radius_m)
    |   movel([0.090194, -1.273895, -2.598735, -0.839759, 1.570796, 1.660990],accel_mss,speed_ms,0,blend_radius_m)
    |   movel([0.090194, -1.300054, -2.612046, -0.800289, 1.570796, 1.660990],accel_mss,speed_ms,0,blend_radius_m)
    |   speed_ms = 0.003
    |   movel([0.090194, -1.310304, -2.616905, -0.785180, 1.570796, 1.660990],accel_mss,speed_ms,0,blend_radius_m)
    |   speed_ms = 0.007
    |   movel([0.091881, -1.308449, -2.618033, -0.785907, 1.570796, 1.662678],accel_mss,speed_ms,0,blend_radius_m)
    |   movel([0.093261, -1.307710, -2.618481, -0.786198, 1.570796, 1.664057],accel_mss,speed_ms,0,blend_radius_m)
    |   movel([0.094545, -1.307450, -2.618639, -0.786300, 1.570796, 1.665342],accel_mss,speed_ms,0,blend_radius_m)
    |   movel([0.095586, -1.307711, -2.618480, -0.786197, 1.570796, 1.666383],accel_mss,speed_ms,0,blend_radius_m)
    |   movel([0.096268, -1.308456, -2.618029, -0.785904, 1.570796, 1.667065],accel_mss,speed_ms,0,blend_radius_m)
    |   movel([0.096402, -1.308965, -2.617719, -0.785704, 1.570796, 1.667198],accel_mss,speed_ms,0,blend_radius_m)
    |   movel([0.096383, -1.309618, -2.617323, -0.785449, 1.570796, 1.667179],accel_mss,speed_ms,0,blend_radius_m)
    |   movel([0.096219, -1.310326, -2.616892, -0.785172, 1.570796, 1.667015],accel_mss,speed_ms,0,blend_radius_m)
    |   movel([0.095924, -1.311003, -2.616479, -0.784908, 1.570796, 1.666721],accel_mss,speed_ms,0,blend_radius_m)
    |   movel([0.095337, -1.311867, -2.615950, -0.784571, 1.570796, 1.666134],accel_mss,speed_ms,0,blend_radius_m)
    |   movel([0.094603, -1.312601, -2.615502, -0.784287, 1.570796, 1.665399],accel_mss,speed_ms,0,blend_radius_m)
    |   movel([0.093731, -1.313184, -2.615144, -0.784061, 1.570796, 1.664527],accel_mss,speed_ms,0,blend_radius_m)
    |   movel([0.092744, -1.313607, -2.614885, -0.783897, 1.570796, 1.663540],accel_mss,speed_ms,0,blend_radius_m)
    |   movel([0.090757, -1.313624, -2.614874, -0.783890, 1.570796, 1.661553],accel_mss,speed_ms,0,blend_radius_m)
    |   movel([0.089757, -1.312332, -2.615666, -0.784391, 1.570796, 1.660553],accel_mss,speed_ms,0,blend_radius_m)
    |   movel([0.090194, -1.310304, -2.616905, -0.785180, 1.570796, 1.660990],accel_mss,speed_ms,0,blend_radius_m)
    |   speed_ms = 0.003
    |   movel([0.090194, -1.313774, -2.618508, -0.780107, 1.570796, 1.660990],accel_mss,speed_ms,0,blend_radius_m)
    |   speed_ms = 0.007
    |   movel([0.091881, -1.311924, -2.619639, -0.780826, 1.570796, 1.662678],accel_mss,speed_ms,0,blend_radius_m)
    |   movel([0.093261, -1.311186, -2.620089, -0.781114, 1.570796, 1.664057],accel_mss,speed_ms,0,blend_radius_m)
    |   movel([0.094545, -1.310927, -2.620246, -0.781215, 1.570796, 1.665342],accel_mss,speed_ms,0,blend_radius_m)
    |   movel([0.095586, -1.311188, -2.620088, -0.781113, 1.570796, 1.666383],accel_mss,speed_ms,0,blend_radius_m)
    |   movel([0.096268, -1.311931, -2.619635, -0.780823, 1.570796, 1.667065],accel_mss,speed_ms,0,blend_radius_m)
    |   movel([0.096402, -1.312439, -2.619325, -0.780625, 1.570796, 1.667198],accel_mss,speed_ms,0,blend_radius_m)
    |   movel([0.096383, -1.313090, -2.618927, -0.780372, 1.570796, 1.667179],accel_mss,speed_ms,0,blend_radius_m)
    |   movel([0.096219, -1.313796, -2.618494, -0.780098, 1.570796, 1.667015],accel_mss,speed_ms,0,blend_radius_m)
    |   movel([0.095924, -1.314472, -2.618080, -0.779837, 1.570796, 1.666721],accel_mss,speed_ms,0,blend_radius_m)
    |   movel([0.095337, -1.315334, -2.617551, -0.779504, 1.570796, 1.666134],accel_mss,speed_ms,0,blend_radius_m)
    |   movel([0.094603, -1.316066, -2.617101, -0.779222, 1.570796, 1.665399],accel_mss,speed_ms,0,blend_radius_m)
    |   movel([0.093731, -1.316648, -2.616742, -0.778999, 1.570796, 1.664527],accel_mss,speed_ms,0,blend_radius_m)
    |   movel([0.092744, -1.317070, -2.616482, -0.778837, 1.570796, 1.663540],accel_mss,speed_ms,0,blend_radius_m)
    |   movel([0.090757, -1.317087, -2.616472, -0.778830, 1.570796, 1.661553],accel_mss,speed_ms,0,blend_radius_m)
    |   movel([0.089757, -1.315798, -2.617265, -0.779325, 1.570796, 1.660553],accel_mss,speed_ms,0,blend_radius_m)
    |   movel([0.090194, -1.313774, -2.618508, -0.780107, 1.570796, 1.660990],accel_mss,speed_ms,0,blend_radius_m)
    |   speed_ms = 0.003
    |   movel([0.090194, -1.300054, -2.612046, -0.800289, 1.570796, 1.660990],accel_mss,speed_ms,0,blend_radius_m)
    |   speed_ms = 1.000
    |   movel([0.090194, -1.273895, -2.598735, -0.839759, 1.570796, 1.660990],accel_mss,speed_ms,0,blend_radius_m)
    |   movel([0.074648, -1.283142, -2.593332, -0.835915, 1.570796, 1.645444],accel_mss,speed_ms,0,blend_radius_m)
    |   movel([0.074648, -1.309165, -2.606523, -0.796701, 1.570796, 1.645444],accel_mss,speed_ms,0,blend_radius_m)
    |   speed_ms = 0.003
    |   movel([0.074648, -1.319355, -2.611336, -0.781699, 1.570796, 1.645444],accel_mss,speed_ms,0,blend_radius_m)
    |   speed_ms = 0.007
    |   movel([0.074675, -1.319767, -2.611079, -0.781543, 1.570796, 1.645472],accel_mss,speed_ms,0,blend_radius_m)
    |   movel([0.074553, -1.320280, -2.610760, -0.781349, 1.570796, 1.645349],accel_mss,speed_ms,0,blend_radius_m)
    |   movel([0.074440, -1.320583, -2.610571, -0.781234, 1.570796, 1.645237],accel_mss,speed_ms,0,blend_radius_m)
    |   movel([0.074315, -1.320855, -2.610402, -0.781132, 1.570796, 1.645112],accel_mss,speed_ms,0,blend_radius_m)
    |   movel([0.073757, -1.321736, -2.609852, -0.780801, 1.570796, 1.644553],accel_mss,speed_ms,0,blend_radius_m)
    |   movel([0.073104, -1.322417, -2.609427, -0.780545, 1.570796, 1.643900],accel_mss,speed_ms,0,blend_radius_m)
    |   movel([0.072314, -1.322927, -2.609108, -0.780355, 1.570796, 1.643111],accel_mss,speed_ms,0,blend_radius_m)
    |   movel([0.071362, -1.323294, -2.608878, -0.780217, 1.570796, 1.642159],accel_mss,speed_ms,0,blend_radius_m)
    |   movel([0.070869, -1.323423, -2.608797, -0.780169, 1.570796, 1.641665],accel_mss,speed_ms,0,blend_radius_m)
    |   movel([0.070526, -1.323474, -2.608765, -0.780150, 1.570796, 1.641322],accel_mss,speed_ms,0,blend_radius_m)
    |   movel([0.070234, -1.323465, -2.608771, -0.780154, 1.570796, 1.641030],accel_mss,speed_ms,0,blend_radius_m)
    |   movel([0.069916, -1.323397, -2.608813, -0.780179, 1.570796, 1.640712],accel_mss,speed_ms,0,blend_radius_m)
    |   movel([0.069099, -1.322793, -2.609191, -0.780404, 1.570796, 1.639896],accel_mss,speed_ms,0,blend_radius_m)
    |   movel([0.068874, -1.321709, -2.609869, -0.780811, 1.570796, 1.639671],accel_mss,speed_ms,0,blend_radius_m)
    |   movel([0.069290, -1.320407, -2.610681, -0.781301, 1.570796, 1.640086],accel_mss,speed_ms,0,blend_radius_m)
    |   movel([0.070255, -1.319201, -2.611431, -0.781757, 1.570796, 1.641051],accel_mss,speed_ms,0,blend_radius_m)
    |   movel([0.070604, -1.318907, -2.611613, -0.781868, 1.570796, 1.641400],accel_mss,speed_ms,0,blend_radius_m)
    |   movel([0.070915, -1.318695, -2.611745, -0.781949, 1.570796, 1.641711],accel_mss,speed_ms,0,blend_radius_m)
    |   movel([0.071271, -1.318512, -2.611859, -0.782018, 1.570796, 1.642068],accel_mss,speed_ms,0,blend_radius_m)
    |   movel([0.071774, -1.318306, -2.611986, -0.782096, 1.570796, 1.642570],accel_mss,speed_ms,0,blend_radius_m)
    |   movel([0.072472, -1.318085, -2.612123, -0.782180, 1.570796, 1.643268],accel_mss,speed_ms,0,blend_radius_m)
    |   movel([0.073056, -1.318004, -2.612174, -0.782212, 1.570796, 1.643852],accel_mss,speed_ms,0,blend_radius_m)
    |   movel([0.073553, -1.318057, -2.612141, -0.782191, 1.570796, 1.644349],accel_mss,speed_ms,0,blend_radius_m)
    |   movel([0.073982, -1.318249, -2.612022, -0.782118, 1.570796, 1.644779],accel_mss,speed_ms,0,blend_radius_m)
    |   movel([0.074267, -1.318512, -2.611859, -0.782018, 1.570796, 1.645063],accel_mss,speed_ms,0,blend_radius_m)
    |   movel([0.074500, -1.318909, -2.611612, -0.781868, 1.570796, 1.645296],accel_mss,speed_ms,0,blend_radius_m)
    |   movel([0.074648, -1.319355, -2.611336, -0.781699, 1.570796, 1.645444],accel_mss,speed_ms,0,blend_radius_m)
    |   speed_ms = 0.003
    |   movel([0.074648, -1.322804, -2.612923, -0.776662, 1.570796, 1.645444],accel_mss,speed_ms,0,blend_radius_m)
    |   speed_ms = 0.007
    |   movel([0.074675, -1.323216, -2.612666, -0.776507, 1.570796, 1.645472],accel_mss,speed_ms,0,blend_radius_m)
    |   movel([0.074553, -1.323727, -2.612346, -0.776316, 1.570796, 1.645349],accel_mss,speed_ms,0,blend_radius_m)
    |   movel([0.074440, -1.324030, -2.612157, -0.776203, 1.570796, 1.645237],accel_mss,speed_ms,0,blend_radius_m)
    |   movel([0.074315, -1.324301, -2.611987, -0.776101, 1.570796, 1.645112],accel_mss,speed_ms,0,blend_radius_m)
    |   movel([0.073757, -1.325180, -2.611436, -0.775773, 1.570796, 1.644553],accel_mss,speed_ms,0,blend_radius_m)
    |   movel([0.073104, -1.325859, -2.611009, -0.775521, 1.570796, 1.643900],accel_mss,speed_ms,0,blend_radius_m)
    |   movel([0.072314, -1.326368, -2.610689, -0.775332, 1.570796, 1.643111],accel_mss,speed_ms,0,blend_radius_m)
    |   movel([0.071362, -1.326734, -2.610459, -0.775196, 1.570796, 1.642159],accel_mss,speed_ms,0,blend_radius_m)
    |   movel([0.070869, -1.326862, -2.610378, -0.775149, 1.570796, 1.641665],accel_mss,speed_ms,0,blend_radius_m)
    |   movel([0.070526, -1.326913, -2.610346, -0.775130, 1.570796, 1.641322],accel_mss,speed_ms,0,blend_radius_m)
    |   movel([0.070234, -1.326904, -2.610351, -0.775133, 1.570796, 1.641030],accel_mss,speed_ms,0,blend_radius_m)
    |   movel([0.069916, -1.326837, -2.610394, -0.775159, 1.570796, 1.640712],accel_mss,speed_ms,0,blend_radius_m)
    |   movel([0.069099, -1.326234, -2.610773, -0.775382, 1.570796, 1.639896],accel_mss,speed_ms,0,blend_radius_m)
    |   movel([0.068874, -1.325153, -2.611453, -0.775784, 1.570796, 1.639671],accel_mss,speed_ms,0,blend_radius_m)
    |   movel([0.069290, -1.323854, -2.612267, -0.776268, 1.570796, 1.640086],accel_mss,speed_ms,0,blend_radius_m)
    |   movel([0.070255, -1.322650, -2.613019, -0.776720, 1.570796, 1.641051],accel_mss,speed_ms,0,blend_radius_m)
    |   movel([0.070604, -1.322358, -2.613202, -0.776829, 1.570796, 1.641400],accel_mss,speed_ms,0,blend_radius_m)
    |   movel([0.070915, -1.322146, -2.613334, -0.776909, 1.570796, 1.641711],accel_mss,speed_ms,0,blend_radius_m)
    |   movel([0.071271, -1.321963, -2.613448, -0.776978, 1.570796, 1.642068],accel_mss,speed_ms,0,blend_radius_m)
    |   movel([0.071774, -1.321758, -2.613576, -0.777055, 1.570796, 1.642570],accel_mss,speed_ms,0,blend_radius_m)
    |   movel([0.072472, -1.321538, -2.613713, -0.777138, 1.570796, 1.643268],accel_mss,speed_ms,0,blend_radius_m)
    |   movel([0.073056, -1.321456, -2.613764, -0.777169, 1.570796, 1.643852],accel_mss,speed_ms,0,blend_radius_m)
    |   movel([0.073553, -1.321509, -2.613731, -0.777149, 1.570796, 1.644349],accel_mss,speed_ms,0,blend_radius_m)
    |   movel([0.073982, -1.321701, -2.613611, -0.777077, 1.570796, 1.644779],accel_mss,speed_ms,0,blend_radius_m)
    |   movel([0.074267, -1.321963, -2.613448, -0.776978, 1.570796, 1.645063],accel_mss,speed_ms,0,blend_radius_m)
    |   movel([0.074500, -1.322359, -2.613201, -0.776829, 1.570796, 1.645296],accel_mss,speed_ms,0,blend_radius_m)
    |   movel([0.074648, -1.322804, -2.612923, -0.776662, 1.570796, 1.645444],accel_mss,speed_ms,0,blend_radius_m)
    |   speed_ms = 0.003
    |   movel([0.074648, -1.309165, -2.606523, -0.796701, 1.570796, 1.645444],accel_mss,speed_ms,0,blend_radius_m)
    |   speed_ms = 1.000
    |   movel([0.074648, -1.283142, -2.593332, -0.835915, 1.570796, 1.645444],accel_mss,speed_ms,0,blend_radius_m)
    |   movel([0.075024, -1.282687, -2.593600, -0.836102, 1.570796, 1.645820],accel_mss,speed_ms,0,blend_radius_m)
    |   movel([0.075024, -1.308718, -2.606796, -0.796875, 1.570796, 1.645820],accel_mss,speed_ms,0,blend_radius_m)
    |   speed_ms = 0.003
    |   movel([0.075024, -1.318910, -2.611612, -0.781867, 1.570796, 1.645820],accel_mss,speed_ms,0,blend_radius_m)
    |   speed_ms = 0.007
    |   movel([0.075085, -1.319510, -2.611239, -0.781640, 1.570796, 1.645881],accel_mss,speed_ms,0,blend_radius_m)
    |   movel([0.074948, -1.320246, -2.610781, -0.781362, 1.570796, 1.645744],accel_mss,speed_ms,0,blend_radius_m)
    |   movel([0.074641, -1.321022, -2.610298, -0.781069, 1.570796, 1.645437],accel_mss,speed_ms,0,blend_radius_m)
    |   movel([0.074198, -1.321742, -2.609848, -0.780798, 1.570796, 1.644994],accel_mss,speed_ms,0,blend_radius_m)
    |   movel([0.073687, -1.322309, -2.609494, -0.780586, 1.570796, 1.644483],accel_mss,speed_ms,0,blend_radius_m)
    |   movel([0.073025, -1.322849, -2.609156, -0.780384, 1.570796, 1.643822],accel_mss,speed_ms,0,blend_radius_m)
    |   movel([0.072291, -1.323304, -2.608871, -0.780213, 1.570796, 1.643087],accel_mss,speed_ms,0,blend_radius_m)
    |   movel([0.071565, -1.323618, -2.608674, -0.780096, 1.570796, 1.642362],accel_mss,speed_ms,0,blend_radius_m)
    |   movel([0.070602, -1.323847, -2.608531, -0.780011, 1.570796, 1.641398],accel_mss,speed_ms,0,blend_radius_m)
    |   movel([0.069813, -1.323830, -2.608542, -0.780017, 1.570796, 1.640609],accel_mss,speed_ms,0,blend_radius_m)
    |   movel([0.069187, -1.323555, -2.608714, -0.780120, 1.570796, 1.639984],accel_mss,speed_ms,0,blend_radius_m)
    |   movel([0.068697, -1.323026, -2.609045, -0.780317, 1.570796, 1.639493],accel_mss,speed_ms,0,blend_radius_m)
    |   movel([0.068546, -1.322743, -2.609223, -0.780423, 1.570796, 1.639343],accel_mss,speed_ms,0,blend_radius_m)
    |   movel([0.068478, -1.322487, -2.609383, -0.780519, 1.570796, 1.639274],accel_mss,speed_ms,0,blend_radius_m)
    |   movel([0.068472, -1.322167, -2.609583, -0.780639, 1.570796, 1.639268],accel_mss,speed_ms,0,blend_radius_m)
    |   movel([0.068526, -1.321647, -2.609908, -0.780834, 1.570796, 1.639322],accel_mss,speed_ms,0,blend_radius_m)
    |   movel([0.068607, -1.321120, -2.610237, -0.781032, 1.570796, 1.639403],accel_mss,speed_ms,0,blend_radius_m)
    |   movel([0.068702, -1.320774, -2.610453, -0.781163, 1.570796, 1.639499],accel_mss,speed_ms,0,blend_radius_m)
    |   movel([0.068847, -1.320465, -2.610645, -0.781279, 1.570796, 1.639644],accel_mss,speed_ms,0,blend_radius_m)
    |   movel([0.069093, -1.320085, -2.610882, -0.781423, 1.570796, 1.639889],accel_mss,speed_ms,0,blend_radius_m)
    |   movel([0.069307, -1.319800, -2.611058, -0.781530, 1.570796, 1.640103],accel_mss,speed_ms,0,blend_radius_m)
    |   movel([0.069588, -1.319471, -2.611263, -0.781655, 1.570796, 1.640384],accel_mss,speed_ms,0,blend_radius_m)
    |   movel([0.069884, -1.319150, -2.611463, -0.781776, 1.570796, 1.640680],accel_mss,speed_ms,0,blend_radius_m)
    |   movel([0.070148, -1.318894, -2.611621, -0.781873, 1.570796, 1.640945],accel_mss,speed_ms,0,blend_radius_m)
    |   movel([0.070517, -1.318583, -2.611815, -0.781991, 1.570796, 1.641314],accel_mss,speed_ms,0,blend_radius_m)
    |   movel([0.070837, -1.318370, -2.611946, -0.782072, 1.570796, 1.641633],accel_mss,speed_ms,0,blend_radius_m)
    |   movel([0.071214, -1.318184, -2.612062, -0.782143, 1.570796, 1.642011],accel_mss,speed_ms,0,blend_radius_m)
    |   movel([0.071809, -1.317950, -2.612207, -0.782232, 1.570796, 1.642605],accel_mss,speed_ms,0,blend_radius_m)
    |   movel([0.072379, -1.317746, -2.612333, -0.782309, 1.570796, 1.643176],accel_mss,speed_ms,0,blend_radius_m)
    |   movel([0.072764, -1.317643, -2.612397, -0.782349, 1.570796, 1.643560],accel_mss,speed_ms,0,blend_radius_m)
    |   movel([0.073074, -1.317602, -2.612422, -0.782364, 1.570796, 1.643870],accel_mss,speed_ms,0,blend_radius_m)
    |   movel([0.073396, -1.317616, -2.612414, -0.782359, 1.570796, 1.644192],accel_mss,speed_ms,0,blend_radius_m)
    |   movel([0.073967, -1.317754, -2.612329, -0.782307, 1.570796, 1.644763],accel_mss,speed_ms,0,blend_radius_m)
    |   movel([0.074437, -1.318021, -2.612163, -0.782205, 1.570796, 1.645234],accel_mss,speed_ms,0,blend_radius_m)
    |   movel([0.074794, -1.318414, -2.611920, -0.782056, 1.570796, 1.645591],accel_mss,speed_ms,0,blend_radius_m)
    |   movel([0.075024, -1.318910, -2.611612, -0.781867, 1.570796, 1.645820],accel_mss,speed_ms,0,blend_radius_m)
    |   speed_ms = 0.003
    |   movel([0.075024, -1.322360, -2.613200, -0.776828, 1.570796, 1.645820],accel_mss,speed_ms,0,blend_radius_m)
    |   speed_ms = 0.007
    |   movel([0.075085, -1.322959, -2.612826, -0.776604, 1.570796, 1.645881],accel_mss,speed_ms,0,blend_radius_m)
    |   movel([0.074948, -1.323693, -2.612367, -0.776328, 1.570796, 1.645744],accel_mss,speed_ms,0,blend_radius_m)
    |   movel([0.074641, -1.324467, -2.611883, -0.776039, 1.570796, 1.645437],accel_mss,speed_ms,0,blend_radius_m)
    |   movel([0.074198, -1.325186, -2.611432, -0.775771, 1.570796, 1.644994],accel_mss,speed_ms,0,blend_radius_m)
    |   movel([0.073687, -1.325751, -2.611077, -0.775561, 1.570796, 1.644483],accel_mss,speed_ms,0,blend_radius_m)
    |   movel([0.073025, -1.326290, -2.610738, -0.775361, 1.570796, 1.643822],accel_mss,speed_ms,0,blend_radius_m)
    |   movel([0.072291, -1.326744, -2.610452, -0.775193, 1.570796, 1.643087],accel_mss,speed_ms,0,blend_radius_m)
    |   movel([0.071565, -1.327058, -2.610255, -0.775077, 1.570796, 1.642362],accel_mss,speed_ms,0,blend_radius_m)
    |   movel([0.070602, -1.327285, -2.610111, -0.774992, 1.570796, 1.641398],accel_mss,speed_ms,0,blend_radius_m)
    |   movel([0.069813, -1.327269, -2.610122, -0.774999, 1.570796, 1.640609],accel_mss,speed_ms,0,blend_radius_m)
    |   movel([0.069187, -1.326994, -2.610295, -0.775100, 1.570796, 1.639984],accel_mss,speed_ms,0,blend_radius_m)
    |   movel([0.068697, -1.326467, -2.610627, -0.775296, 1.570796, 1.639493],accel_mss,speed_ms,0,blend_radius_m)
    |   movel([0.068546, -1.326184, -2.610804, -0.775400, 1.570796, 1.639343],accel_mss,speed_ms,0,blend_radius_m)
    |   movel([0.068478, -1.325929, -2.610965, -0.775495, 1.570796, 1.639274],accel_mss,speed_ms,0,blend_radius_m)
    |   movel([0.068472, -1.325610, -2.611166, -0.775614, 1.570796, 1.639268],accel_mss,speed_ms,0,blend_radius_m)
    |   movel([0.068526, -1.325091, -2.611492, -0.775807, 1.570796, 1.639322],accel_mss,speed_ms,0,blend_radius_m)
    |   movel([0.068607, -1.324565, -2.611821, -0.776003, 1.570796, 1.639403],accel_mss,speed_ms,0,blend_radius_m)
    |   movel([0.068702, -1.324220, -2.612038, -0.776132, 1.570796, 1.639499],accel_mss,speed_ms,0,blend_radius_m)
    |   movel([0.068847, -1.323912, -2.612230, -0.776247, 1.570796, 1.639644],accel_mss,speed_ms,0,blend_radius_m)
    |   movel([0.069093, -1.323532, -2.612468, -0.776389, 1.570796, 1.639889],accel_mss,speed_ms,0,blend_radius_m)
    |   movel([0.069307, -1.323249, -2.612645, -0.776495, 1.570796, 1.640103],accel_mss,speed_ms,0,blend_radius_m)
    |   movel([0.069588, -1.322920, -2.612851, -0.776618, 1.570796, 1.640384],accel_mss,speed_ms,0,blend_radius_m)
    |   movel([0.069884, -1.322600, -2.613051, -0.776738, 1.570796, 1.640680],accel_mss,speed_ms,0,blend_radius_m)
    |   movel([0.070148, -1.322345, -2.613210, -0.776834, 1.570796, 1.640945],accel_mss,speed_ms,0,blend_radius_m)
    |   movel([0.070517, -1.322034, -2.613404, -0.776951, 1.570796, 1.641314],accel_mss,speed_ms,0,blend_radius_m)
    |   movel([0.070837, -1.321822, -2.613536, -0.777031, 1.570796, 1.641633],accel_mss,speed_ms,0,blend_radius_m)
    |   movel([0.071214, -1.321636, -2.613652, -0.777101, 1.570796, 1.642011],accel_mss,speed_ms,0,blend_radius_m)
    |   movel([0.071809, -1.321402, -2.613797, -0.777189, 1.570796, 1.642605],accel_mss,speed_ms,0,blend_radius_m)
    |   movel([0.072379, -1.321200, -2.613923, -0.777266, 1.570796, 1.643176],accel_mss,speed_ms,0,blend_radius_m)
    |   movel([0.072764, -1.321096, -2.613988, -0.777305, 1.570796, 1.643560],accel_mss,speed_ms,0,blend_radius_m)
    |   movel([0.073074, -1.321056, -2.614013, -0.777320, 1.570796, 1.643870],accel_mss,speed_ms,0,blend_radius_m)
    |   movel([0.073396, -1.321069, -2.614005, -0.777315, 1.570796, 1.644192],accel_mss,speed_ms,0,blend_radius_m)
    |   movel([0.073967, -1.321207, -2.613919, -0.777263, 1.570796, 1.644763],accel_mss,speed_ms,0,blend_radius_m)
    |   movel([0.074437, -1.321474, -2.613753, -0.777162, 1.570796, 1.645234],accel_mss,speed_ms,0,blend_radius_m)
    |   movel([0.074794, -1.321865, -2.613509, -0.777015, 1.570796, 1.645591],accel_mss,speed_ms,0,blend_radius_m)
    |   movel([0.075024, -1.322360, -2.613200, -0.776828, 1.570796, 1.645820],accel_mss,speed_ms,0,blend_radius_m)
    |   speed_ms = 0.003
    |   movel([0.075024, -1.308718, -2.606796, -0.796875, 1.570796, 1.645820],accel_mss,speed_ms,0,blend_radius_m)
    |   speed_ms = 1.000
    |   movel([0.075024, -1.282687, -2.593600, -0.836102, 1.570796, 1.645820],accel_mss,speed_ms,0,blend_radius_m)
    |   movel([0.074027, -1.283141, -2.593332, -0.835916, 1.570796, 1.644824],accel_mss,speed_ms,0,blend_radius_m)
    |   movel([0.074027, -1.309165, -2.606523, -0.796701, 1.570796, 1.644824],accel_mss,speed_ms,0,blend_radius_m)
    |   speed_ms = 0.003
    |   movel([0.074027, -1.319354, -2.611336, -0.781699, 1.570796, 1.644824],accel_mss,speed_ms,0,blend_radius_m)
    |   speed_ms = 0.007
    |   movel([0.073556, -1.319849, -2.611028, -0.781512, 1.570796, 1.644352],accel_mss,speed_ms,0,blend_radius_m)
    |   movel([0.072865, -1.320341, -2.610722, -0.781326, 1.570796, 1.643661],accel_mss,speed_ms,0,blend_radius_m)
    |   movel([0.072601, -1.320557, -2.610588, -0.781244, 1.570796, 1.643397],accel_mss,speed_ms,0,blend_radius_m)
    |   movel([0.072444, -1.321001, -2.610311, -0.781077, 1.570796, 1.643240],accel_mss,speed_ms,0,blend_radius_m)
    |   movel([0.072443, -1.321758, -2.609838, -0.780792, 1.570796, 1.643239],accel_mss,speed_ms,0,blend_radius_m)
    |   movel([0.072434, -1.321990, -2.609693, -0.780705, 1.570796, 1.643230],accel_mss,speed_ms,0,blend_radius_m)
    |   movel([0.072327, -1.322242, -2.609536, -0.780611, 1.570796, 1.643123],accel_mss,speed_ms,0,blend_radius_m)
    |   movel([0.071996, -1.322298, -2.609501, -0.780590, 1.570796, 1.642792],accel_mss,speed_ms,0,blend_radius_m)
    |   movel([0.071795, -1.321918, -2.609739, -0.780733, 1.570796, 1.642591],accel_mss,speed_ms,0,blend_radius_m)
    |   movel([0.071704, -1.321719, -2.609863, -0.780807, 1.570796, 1.642500],accel_mss,speed_ms,0,blend_radius_m)
    |   movel([0.071601, -1.321544, -2.609972, -0.780873, 1.570796, 1.642397],accel_mss,speed_ms,0,blend_radius_m)
    |   movel([0.071406, -1.321373, -2.610079, -0.780937, 1.570796, 1.642202],accel_mss,speed_ms,0,blend_radius_m)
    |   movel([0.071079, -1.321469, -2.610019, -0.780901, 1.570796, 1.641875],accel_mss,speed_ms,0,blend_radius_m)
    |   movel([0.070562, -1.321740, -2.609850, -0.780799, 1.570796, 1.641358],accel_mss,speed_ms,0,blend_radius_m)
    |   movel([0.070211, -1.321941, -2.609724, -0.780724, 1.570796, 1.641007],accel_mss,speed_ms,0,blend_radius_m)
    |   movel([0.069848, -1.322070, -2.609644, -0.780675, 1.570796, 1.640644],accel_mss,speed_ms,0,blend_radius_m)
    |   movel([0.069610, -1.321995, -2.609690, -0.780703, 1.570796, 1.640407],accel_mss,speed_ms,0,blend_radius_m)
    |   movel([0.069744, -1.321703, -2.609873, -0.780813, 1.570796, 1.640540],accel_mss,speed_ms,0,blend_radius_m)
    |   movel([0.070057, -1.321421, -2.610049, -0.780919, 1.570796, 1.640853],accel_mss,speed_ms,0,blend_radius_m)
    |   movel([0.070500, -1.321122, -2.610236, -0.781032, 1.570796, 1.641296],accel_mss,speed_ms,0,blend_radius_m)
    |   movel([0.070910, -1.320839, -2.610412, -0.781138, 1.570796, 1.641707],accel_mss,speed_ms,0,blend_radius_m)
    |   movel([0.071115, -1.320581, -2.610573, -0.781235, 1.570796, 1.641911],accel_mss,speed_ms,0,blend_radius_m)
    |   movel([0.071162, -1.320290, -2.610754, -0.781345, 1.570796, 1.641958],accel_mss,speed_ms,0,blend_radius_m)
    |   movel([0.071051, -1.319883, -2.611007, -0.781499, 1.570796, 1.641848],accel_mss,speed_ms,0,blend_radius_m)
    |   movel([0.070960, -1.319617, -2.611172, -0.781599, 1.570796, 1.641757],accel_mss,speed_ms,0,blend_radius_m)
    |   movel([0.070970, -1.319306, -2.611366, -0.781717, 1.570796, 1.641766],accel_mss,speed_ms,0,blend_radius_m)
    |   movel([0.071177, -1.319020, -2.611543, -0.781825, 1.570796, 1.641973],accel_mss,speed_ms,0,blend_radius_m)
    |   movel([0.071466, -1.319017, -2.611546, -0.781827, 1.570796, 1.642262],accel_mss,speed_ms,0,blend_radius_m)
    |   movel([0.071655, -1.319206, -2.611428, -0.781755, 1.570796, 1.642451],accel_mss,speed_ms,0,blend_radius_m)
    |   movel([0.071802, -1.319519, -2.611233, -0.781636, 1.570796, 1.642598],accel_mss,speed_ms,0,blend_radius_m)
    |   movel([0.071941, -1.319865, -2.611019, -0.781506, 1.570796, 1.642737],accel_mss,speed_ms,0,blend_radius_m)
    |   movel([0.072115, -1.319984, -2.610944, -0.781461, 1.570796, 1.642911],accel_mss,speed_ms,0,blend_radius_m)
    |   movel([0.072792, -1.319712, -2.611113, -0.781564, 1.570796, 1.643588],accel_mss,speed_ms,0,blend_radius_m)
    |   movel([0.073214, -1.319464, -2.611268, -0.781657, 1.570796, 1.644010],accel_mss,speed_ms,0,blend_radius_m)
    |   movel([0.073566, -1.319296, -2.611372, -0.781721, 1.570796, 1.644362],accel_mss,speed_ms,0,blend_radius_m)
    |   movel([0.073838, -1.319207, -2.611427, -0.781754, 1.570796, 1.644634],accel_mss,speed_ms,0,blend_radius_m)
    |   movel([0.074027, -1.319354, -2.611336, -0.781699, 1.570796, 1.644824],accel_mss,speed_ms,0,blend_radius_m)
    |   speed_ms = 0.003
    |   movel([0.074027, -1.322803, -2.612924, -0.776662, 1.570796, 1.644824],accel_mss,speed_ms,0,blend_radius_m)
    |   speed_ms = 0.007
    |   movel([0.073556, -1.323297, -2.612615, -0.776477, 1.570796, 1.644352],accel_mss,speed_ms,0,blend_radius_m)
    |   movel([0.072865, -1.323788, -2.612308, -0.776293, 1.570796, 1.643661],accel_mss,speed_ms,0,blend_radius_m)
    |   movel([0.072601, -1.324003, -2.612173, -0.776212, 1.570796, 1.643397],accel_mss,speed_ms,0,blend_radius_m)
    |   movel([0.072444, -1.324446, -2.611896, -0.776047, 1.570796, 1.643240],accel_mss,speed_ms,0,blend_radius_m)
    |   movel([0.072443, -1.325202, -2.611422, -0.775765, 1.570796, 1.643239],accel_mss,speed_ms,0,blend_radius_m)
    |   movel([0.072434, -1.325433, -2.611276, -0.775679, 1.570796, 1.643230],accel_mss,speed_ms,0,blend_radius_m)
    |   movel([0.072327, -1.325684, -2.611119, -0.775586, 1.570796, 1.643123],accel_mss,speed_ms,0,blend_radius_m)
    |   movel([0.071996, -1.325740, -2.611084, -0.775565, 1.570796, 1.642792],accel_mss,speed_ms,0,blend_radius_m)
    |   movel([0.071795, -1.325361, -2.611322, -0.775706, 1.570796, 1.642591],accel_mss,speed_ms,0,blend_radius_m)
    |   movel([0.071704, -1.325162, -2.611447, -0.775780, 1.570796, 1.642500],accel_mss,speed_ms,0,blend_radius_m)
    |   movel([0.071601, -1.324988, -2.611556, -0.775845, 1.570796, 1.642397],accel_mss,speed_ms,0,blend_radius_m)
    |   movel([0.071406, -1.324817, -2.611663, -0.775908, 1.570796, 1.642202],accel_mss,speed_ms,0,blend_radius_m)
    |   movel([0.071079, -1.324913, -2.611603, -0.775873, 1.570796, 1.641875],accel_mss,speed_ms,0,blend_radius_m)
    |   movel([0.070562, -1.325183, -2.611434, -0.775772, 1.570796, 1.641358],accel_mss,speed_ms,0,blend_radius_m)
    |   movel([0.070211, -1.325384, -2.611307, -0.775697, 1.570796, 1.641007],accel_mss,speed_ms,0,blend_radius_m)
    |   movel([0.069848, -1.325513, -2.611227, -0.775650, 1.570796, 1.640644],accel_mss,speed_ms,0,blend_radius_m)
    |   movel([0.069610, -1.325438, -2.611273, -0.775677, 1.570796, 1.640407],accel_mss,speed_ms,0,blend_radius_m)
    |   movel([0.069744, -1.325147, -2.611456, -0.775786, 1.570796, 1.640540],accel_mss,speed_ms,0,blend_radius_m)
    |   movel([0.070057, -1.324865, -2.611633, -0.775891, 1.570796, 1.640853],accel_mss,speed_ms,0,blend_radius_m)
    |   movel([0.070500, -1.324567, -2.611820, -0.776002, 1.570796, 1.641296],accel_mss,speed_ms,0,blend_radius_m)
    |   movel([0.070910, -1.324284, -2.611997, -0.776107, 1.570796, 1.641707],accel_mss,speed_ms,0,blend_radius_m)
    |   movel([0.071115, -1.324028, -2.612158, -0.776203, 1.570796, 1.641911],accel_mss,speed_ms,0,blend_radius_m)
    |   movel([0.071162, -1.323737, -2.612340, -0.776312, 1.570796, 1.641958],accel_mss,speed_ms,0,blend_radius_m)
    |   movel([0.071051, -1.323331, -2.612594, -0.776464, 1.570796, 1.641848],accel_mss,speed_ms,0,blend_radius_m)
    |   movel([0.070960, -1.323066, -2.612759, -0.776563, 1.570796, 1.641757],accel_mss,speed_ms,0,blend_radius_m)
    |   movel([0.070970, -1.322756, -2.612953, -0.776680, 1.570796, 1.641766],accel_mss,speed_ms,0,blend_radius_m)
    |   movel([0.071177, -1.322470, -2.613132, -0.776787, 1.570796, 1.641973],accel_mss,speed_ms,0,blend_radius_m)
    |   movel([0.071466, -1.322467, -2.613134, -0.776789, 1.570796, 1.642262],accel_mss,speed_ms,0,blend_radius_m)
    |   movel([0.071655, -1.322656, -2.613016, -0.776717, 1.570796, 1.642451],accel_mss,speed_ms,0,blend_radius_m)
    |   movel([0.071802, -1.322968, -2.612821, -0.776600, 1.570796, 1.642598],accel_mss,speed_ms,0,blend_radius_m)
    |   movel([0.071941, -1.323313, -2.612605, -0.776471, 1.570796, 1.642737],accel_mss,speed_ms,0,blend_radius_m)
    |   movel([0.072115, -1.323432, -2.612531, -0.776426, 1.570796, 1.642911],accel_mss,speed_ms,0,blend_radius_m)
    |   movel([0.072792, -1.323160, -2.612701, -0.776528, 1.570796, 1.643588],accel_mss,speed_ms,0,blend_radius_m)
    |   movel([0.073214, -1.322913, -2.612855, -0.776621, 1.570796, 1.644010],accel_mss,speed_ms,0,blend_radius_m)
    |   movel([0.073566, -1.322746, -2.612960, -0.776684, 1.570796, 1.644362],accel_mss,speed_ms,0,blend_radius_m)
    |   movel([0.073838, -1.322657, -2.613015, -0.776717, 1.570796, 1.644634],accel_mss,speed_ms,0,blend_radius_m)
    |   movel([0.074027, -1.322803, -2.612924, -0.776662, 1.570796, 1.644824],accel_mss,speed_ms,0,blend_radius_m)
    |   speed_ms = 0.003
    |   movel([0.074027, -1.309165, -2.606523, -0.796701, 1.570796, 1.644824],accel_mss,speed_ms,0,blend_radius_m)
    |   speed_ms = 1.000
    |   movel([0.074027, -1.283141, -2.593332, -0.835916, 1.570796, 1.644824],accel_mss,speed_ms,0,blend_radius_m)
    |   movel([0.071023, -1.278128, -2.596274, -0.837987, 1.570796, 1.641819],accel_mss,speed_ms,0,blend_radius_m)
    |   movel([0.071023, -1.304226, -2.609531, -0.798633, 1.570796, 1.641819],accel_mss,speed_ms,0,blend_radius_m)
    |   speed_ms = 0.003
    |   movel([0.071023, -1.314448, -2.614368, -0.783573, 1.570796, 1.641819],accel_mss,speed_ms,0,blend_radius_m)
    |   speed_ms = 0.007
    |   movel([0.069147, -1.315811, -2.613529, -0.783049, 1.570796, 1.639943],accel_mss,speed_ms,0,blend_radius_m)
    |   movel([0.068357, -1.316304, -2.613225, -0.782860, 1.570796, 1.639153],accel_mss,speed_ms,0,blend_radius_m)
    |   movel([0.067918, -1.316419, -2.613154, -0.782816, 1.570796, 1.638715],accel_mss,speed_ms,0,blend_radius_m)
    |   movel([0.067617, -1.316265, -2.613249, -0.782875, 1.570796, 1.638413],accel_mss,speed_ms,0,blend_radius_m)
    |   movel([0.067573, -1.316019, -2.613400, -0.782969, 1.570796, 1.638369],accel_mss,speed_ms,0,blend_radius_m)
    |   movel([0.067713, -1.315740, -2.613573, -0.783076, 1.570796, 1.638510],accel_mss,speed_ms,0,blend_radius_m)
    |   movel([0.068093, -1.315373, -2.613799, -0.783217, 1.570796, 1.638889],accel_mss,speed_ms,0,blend_radius_m)
    |   movel([0.068839, -1.314811, -2.614145, -0.783433, 1.570796, 1.639635],accel_mss,speed_ms,0,blend_radius_m)
    |   movel([0.070239, -1.313837, -2.614744, -0.783808, 1.570796, 1.641035],accel_mss,speed_ms,0,blend_radius_m)
    |   movel([0.070997, -1.313439, -2.614988, -0.783962, 1.570796, 1.641793],accel_mss,speed_ms,0,blend_radius_m)
    |   movel([0.071373, -1.313456, -2.614977, -0.783955, 1.570796, 1.642169],accel_mss,speed_ms,0,blend_radius_m)
    |   movel([0.071504, -1.313791, -2.614772, -0.783826, 1.570796, 1.642300],accel_mss,speed_ms,0,blend_radius_m)
    |   movel([0.071385, -1.314116, -2.614572, -0.783701, 1.570796, 1.642181],accel_mss,speed_ms,0,blend_radius_m)
    |   movel([0.071023, -1.314448, -2.614368, -0.783573, 1.570796, 1.641819],accel_mss,speed_ms,0,blend_radius_m)
    |   speed_ms = 0.003
    |   movel([0.071023, -1.317909, -2.615964, -0.778516, 1.570796, 1.641819],accel_mss,speed_ms,0,blend_radius_m)
    |   speed_ms = 0.007
    |   movel([0.069147, -1.319269, -2.615122, -0.777998, 1.570796, 1.639943],accel_mss,speed_ms,0,blend_radius_m)
    |   movel([0.068357, -1.319761, -2.614817, -0.777811, 1.570796, 1.639153],accel_mss,speed_ms,0,blend_radius_m)
    |   movel([0.067918, -1.319875, -2.614746, -0.777767, 1.570796, 1.638715],accel_mss,speed_ms,0,blend_radius_m)
    |   movel([0.067617, -1.319722, -2.614841, -0.777825, 1.570796, 1.638413],accel_mss,speed_ms,0,blend_radius_m)
    |   movel([0.067573, -1.319477, -2.614994, -0.777919, 1.570796, 1.638369],accel_mss,speed_ms,0,blend_radius_m)
    |   movel([0.067713, -1.319198, -2.615166, -0.778024, 1.570796, 1.638510],accel_mss,speed_ms,0,blend_radius_m)
    |   movel([0.068093, -1.318831, -2.615394, -0.778164, 1.570796, 1.638889],accel_mss,speed_ms,0,blend_radius_m)
    |   movel([0.068839, -1.318271, -2.615740, -0.778378, 1.570796, 1.639635],accel_mss,speed_ms,0,blend_radius_m)
    |   movel([0.070239, -1.317299, -2.616341, -0.778749, 1.570796, 1.641035],accel_mss,speed_ms,0,blend_radius_m)
    |   movel([0.070997, -1.316902, -2.616586, -0.778901, 1.570796, 1.641793],accel_mss,speed_ms,0,blend_radius_m)
    |   movel([0.071373, -1.316919, -2.616575, -0.778895, 1.570796, 1.642169],accel_mss,speed_ms,0,blend_radius_m)
    |   movel([0.071504, -1.317253, -2.616369, -0.778767, 1.570796, 1.642300],accel_mss,speed_ms,0,blend_radius_m)
    |   movel([0.071385, -1.317578, -2.616169, -0.778642, 1.570796, 1.642181],accel_mss,speed_ms,0,blend_radius_m)
    |   movel([0.071023, -1.317909, -2.615964, -0.778516, 1.570796, 1.641819],accel_mss,speed_ms,0,blend_radius_m)
    |   speed_ms = 0.003
    |   movel([0.071023, -1.304226, -2.609531, -0.798633, 1.570796, 1.641819],accel_mss,speed_ms,0,blend_radius_m)
    |   speed_ms = 1.000
    |   movel([0.071023, -1.278128, -2.596274, -0.837987, 1.570796, 1.641819],accel_mss,speed_ms,0,blend_radius_m)
    |   movel([0.070234, -1.277001, -2.596932, -0.838457, 1.570796, 1.641030],accel_mss,speed_ms,0,blend_radius_m)
    |   movel([0.070234, -1.303115, -2.610203, -0.799072, 1.570796, 1.641030],accel_mss,speed_ms,0,blend_radius_m)
    |   speed_ms = 0.003
    |   movel([0.070234, -1.313344, -2.615046, -0.783999, 1.570796, 1.641030],accel_mss,speed_ms,0,blend_radius_m)
    |   speed_ms = 0.007
    |   movel([0.069690, -1.313736, -2.614806, -0.783847, 1.570796, 1.640486],accel_mss,speed_ms,0,blend_radius_m)
    |   movel([0.069350, -1.313960, -2.614668, -0.783761, 1.570796, 1.640146],accel_mss,speed_ms,0,blend_radius_m)
    |   movel([0.068982, -1.314205, -2.614518, -0.783667, 1.570796, 1.639778],accel_mss,speed_ms,0,blend_radius_m)
    |   movel([0.068608, -1.314463, -2.614359, -0.783567, 1.570796, 1.639404],accel_mss,speed_ms,0,blend_radius_m)
    |   movel([0.068272, -1.314701, -2.614212, -0.783475, 1.570796, 1.639068],accel_mss,speed_ms,0,blend_radius_m)
    |   movel([0.067748, -1.315091, -2.613973, -0.783325, 1.570796, 1.638544],accel_mss,speed_ms,0,blend_radius_m)
    |   movel([0.067368, -1.315127, -2.613951, -0.783312, 1.570796, 1.638164],accel_mss,speed_ms,0,blend_radius_m)
    |   movel([0.067208, -1.314950, -2.614059, -0.783379, 1.570796, 1.638004],accel_mss,speed_ms,0,blend_radius_m)
    |   movel([0.067125, -1.314520, -2.614324, -0.783545, 1.570796, 1.637921],accel_mss,speed_ms,0,blend_radius_m)
    |   movel([0.067331, -1.314004, -2.614641, -0.783744, 1.570796, 1.638127],accel_mss,speed_ms,0,blend_radius_m)
    |   movel([0.067860, -1.313393, -2.615016, -0.783980, 1.570796, 1.638656],accel_mss,speed_ms,0,blend_radius_m)
    |   movel([0.068714, -1.312682, -2.615452, -0.784255, 1.570796, 1.639510],accel_mss,speed_ms,0,blend_radius_m)
    |   movel([0.069595, -1.312087, -2.615816, -0.784486, 1.570796, 1.640391],accel_mss,speed_ms,0,blend_radius_m)
    |   movel([0.070212, -1.311846, -2.615963, -0.784579, 1.570796, 1.641008],accel_mss,speed_ms,0,blend_radius_m)
    |   movel([0.070613, -1.311926, -2.615915, -0.784548, 1.570796, 1.641409],accel_mss,speed_ms,0,blend_radius_m)
    |   movel([0.070831, -1.312303, -2.615684, -0.784402, 1.570796, 1.641627],accel_mss,speed_ms,0,blend_radius_m)
    |   movel([0.070900, -1.312683, -2.615452, -0.784255, 1.570796, 1.641697],accel_mss,speed_ms,0,blend_radius_m)
    |   movel([0.070811, -1.312966, -2.615278, -0.784145, 1.570796, 1.641607],accel_mss,speed_ms,0,blend_radius_m)
    |   movel([0.070439, -1.313152, -2.615164, -0.784073, 1.570796, 1.641236],accel_mss,speed_ms,0,blend_radius_m)
    |   speed_ms = 0.003
    |   movel([0.070234, -1.316808, -2.616644, -0.778937, 1.570796, 1.641030],accel_mss,speed_ms,0,blend_radius_m)
    |   speed_ms = 0.007
    |   movel([0.069690, -1.317199, -2.616403, -0.778788, 1.570796, 1.640486],accel_mss,speed_ms,0,blend_radius_m)
    |   movel([0.069350, -1.317422, -2.616265, -0.778702, 1.570796, 1.640146],accel_mss,speed_ms,0,blend_radius_m)
    |   movel([0.068982, -1.317666, -2.616114, -0.778609, 1.570796, 1.639778],accel_mss,speed_ms,0,blend_radius_m)
    |   movel([0.068608, -1.317924, -2.615955, -0.778510, 1.570796, 1.639404],accel_mss,speed_ms,0,blend_radius_m)
    |   movel([0.068272, -1.318162, -2.615808, -0.778419, 1.570796, 1.639068],accel_mss,speed_ms,0,blend_radius_m)
    |   movel([0.067748, -1.318551, -2.615567, -0.778271, 1.570796, 1.638544],accel_mss,speed_ms,0,blend_radius_m)
    |   movel([0.067368, -1.318586, -2.615545, -0.778257, 1.570796, 1.638164],accel_mss,speed_ms,0,blend_radius_m)
    |   movel([0.067208, -1.318410, -2.615654, -0.778325, 1.570796, 1.638004],accel_mss,speed_ms,0,blend_radius_m)
    |   movel([0.067125, -1.317980, -2.615920, -0.778489, 1.570796, 1.637921],accel_mss,speed_ms,0,blend_radius_m)
    |   movel([0.067331, -1.317466, -2.616238, -0.778685, 1.570796, 1.638127],accel_mss,speed_ms,0,blend_radius_m)
    |   movel([0.067860, -1.316857, -2.616614, -0.778919, 1.570796, 1.638656],accel_mss,speed_ms,0,blend_radius_m)
    |   movel([0.068714, -1.316147, -2.617051, -0.779191, 1.570796, 1.639510],accel_mss,speed_ms,0,blend_radius_m)
    |   movel([0.069595, -1.315553, -2.617416, -0.779420, 1.570796, 1.640391],accel_mss,speed_ms,0,blend_radius_m)
    |   movel([0.070212, -1.315313, -2.617564, -0.779512, 1.570796, 1.641008],accel_mss,speed_ms,0,blend_radius_m)
    |   movel([0.070613, -1.315393, -2.617515, -0.779481, 1.570796, 1.641409],accel_mss,speed_ms,0,blend_radius_m)
    |   movel([0.070831, -1.315769, -2.617283, -0.779336, 1.570796, 1.641627],accel_mss,speed_ms,0,blend_radius_m)
    |   movel([0.070900, -1.316148, -2.617050, -0.779191, 1.570796, 1.641697],accel_mss,speed_ms,0,blend_radius_m)
    |   movel([0.070811, -1.316431, -2.616876, -0.779082, 1.570796, 1.641607],accel_mss,speed_ms,0,blend_radius_m)
    |   movel([0.070439, -1.316616, -2.616762, -0.779011, 1.570796, 1.641236],accel_mss,speed_ms,0,blend_radius_m)
    |   speed_ms = 0.003
    |   movel([0.070234, -1.303115, -2.610203, -0.799072, 1.570796, 1.641030],accel_mss,speed_ms,0,blend_radius_m)
    |   speed_ms = 1.000
    |   movel([0.070234, -1.277001, -2.596932, -0.838457, 1.570796, 1.641030],accel_mss,speed_ms,0,blend_radius_m)
    |   movel([0.073982, -1.263429, -2.604724, -0.844235, 1.570796, 1.644779],accel_mss,speed_ms,0,blend_radius_m)
    |   movel([0.073982, -1.289735, -2.618173, -0.804481, 1.570796, 1.644779],accel_mss,speed_ms,0,blend_radius_m)
    |   speed_ms = 0.003
    |   movel([0.073982, -1.300051, -2.623084, -0.789254, 1.570796, 1.644779],accel_mss,speed_ms,0,blend_radius_m)
    |   speed_ms = 0.007
    |   movel([0.073932, -1.299789, -2.623240, -0.789360, 1.570796, 1.644728],accel_mss,speed_ms,0,blend_radius_m)
    |   movel([0.074261, -1.299549, -2.623383, -0.789457, 1.570796, 1.645057],accel_mss,speed_ms,0,blend_radius_m)
    |   movel([0.074673, -1.299325, -2.623517, -0.789548, 1.570796, 1.645470],accel_mss,speed_ms,0,blend_radius_m)
    |   movel([0.074331, -1.299356, -2.623498, -0.789535, 1.570796, 1.645127],accel_mss,speed_ms,0,blend_radius_m)
    |   movel([0.073782, -1.299594, -2.623356, -0.789439, 1.570796, 1.644579],accel_mss,speed_ms,0,blend_radius_m)
    |   movel([0.072985, -1.299872, -2.623191, -0.789326, 1.570796, 1.643781],accel_mss,speed_ms,0,blend_radius_m)
    |   movel([0.072179, -1.300125, -2.623040, -0.789224, 1.570796, 1.642975],accel_mss,speed_ms,0,blend_radius_m)
    |   movel([0.071902, -1.300103, -2.623053, -0.789233, 1.570796, 1.642698],accel_mss,speed_ms,0,blend_radius_m)
    |   movel([0.071682, -1.300397, -2.622877, -0.789114, 1.570796, 1.642478],accel_mss,speed_ms,0,blend_radius_m)
    |   movel([0.071302, -1.300592, -2.622761, -0.789035, 1.570796, 1.642098],accel_mss,speed_ms,0,blend_radius_m)
    |   movel([0.071480, -1.300308, -2.622931, -0.789150, 1.570796, 1.642277],accel_mss,speed_ms,0,blend_radius_m)
    |   movel([0.071194, -1.300365, -2.622897, -0.789127, 1.570796, 1.641991],accel_mss,speed_ms,0,blend_radius_m)
    |   movel([0.070917, -1.300543, -2.622791, -0.789055, 1.570796, 1.641714],accel_mss,speed_ms,0,blend_radius_m)
    |   movel([0.070724, -1.300383, -2.622886, -0.789120, 1.570796, 1.641520],accel_mss,speed_ms,0,blend_radius_m)
    |   movel([0.070555, -1.300212, -2.622988, -0.789189, 1.570796, 1.641352],accel_mss,speed_ms,0,blend_radius_m)
    |   movel([0.070266, -1.300204, -2.622993, -0.789192, 1.570796, 1.641063],accel_mss,speed_ms,0,blend_radius_m)
    |   movel([0.070498, -1.300295, -2.622938, -0.789155, 1.570796, 1.641294],accel_mss,speed_ms,0,blend_radius_m)
    |   movel([0.070207, -1.300506, -2.622813, -0.789070, 1.570796, 1.641004],accel_mss,speed_ms,0,blend_radius_m)
    |   movel([0.069999, -1.300433, -2.622856, -0.789100, 1.570796, 1.640795],accel_mss,speed_ms,0,blend_radius_m)
    |   movel([0.069864, -1.300276, -2.622950, -0.789163, 1.570796, 1.640660],accel_mss,speed_ms,0,blend_radius_m)
    |   movel([0.069616, -1.300492, -2.622821, -0.789076, 1.570796, 1.640412],accel_mss,speed_ms,0,blend_radius_m)
    |   movel([0.069394, -1.300421, -2.622863, -0.789105, 1.570796, 1.640190],accel_mss,speed_ms,0,blend_radius_m)
    |   movel([0.069164, -1.300073, -2.623071, -0.789245, 1.570796, 1.639960],accel_mss,speed_ms,0,blend_radius_m)
    |   movel([0.068809, -1.300112, -2.623048, -0.789229, 1.570796, 1.639606],accel_mss,speed_ms,0,blend_radius_m)
    |   movel([0.068472, -1.300176, -2.623010, -0.789204, 1.570796, 1.639268],accel_mss,speed_ms,0,blend_radius_m)
    |   movel([0.068228, -1.300130, -2.623037, -0.789222, 1.570796, 1.639025],accel_mss,speed_ms,0,blend_radius_m)
    |   movel([0.068160, -1.299903, -2.623172, -0.789314, 1.570796, 1.638957],accel_mss,speed_ms,0,blend_radius_m)
    |   movel([0.067957, -1.299756, -2.623260, -0.789373, 1.570796, 1.638753],accel_mss,speed_ms,0,blend_radius_m)
    |   movel([0.067920, -1.299501, -2.623411, -0.789476, 1.570796, 1.638717],accel_mss,speed_ms,0,blend_radius_m)
    |   movel([0.068076, -1.299095, -2.623653, -0.789641, 1.570796, 1.638872],accel_mss,speed_ms,0,blend_radius_m)
    |   movel([0.068245, -1.298825, -2.623814, -0.789750, 1.570796, 1.639041],accel_mss,speed_ms,0,blend_radius_m)
    |   movel([0.068538, -1.298372, -2.624083, -0.789934, 1.570796, 1.639334],accel_mss,speed_ms,0,blend_radius_m)
    |   movel([0.068564, -1.298071, -2.624261, -0.790056, 1.570796, 1.639361],accel_mss,speed_ms,0,blend_radius_m)
    |   movel([0.068351, -1.297911, -2.624356, -0.790122, 1.570796, 1.639147],accel_mss,speed_ms,0,blend_radius_m)
    |   movel([0.068159, -1.297750, -2.624452, -0.790187, 1.570796, 1.638955],accel_mss,speed_ms,0,blend_radius_m)
    |   movel([0.068070, -1.297551, -2.624570, -0.790268, 1.570796, 1.638866],accel_mss,speed_ms,0,blend_radius_m)
    |   movel([0.067838, -1.297444, -2.624633, -0.790312, 1.570796, 1.638635],accel_mss,speed_ms,0,blend_radius_m)
    |   movel([0.067733, -1.297246, -2.624751, -0.790392, 1.570796, 1.638529],accel_mss,speed_ms,0,blend_radius_m)
    |   movel([0.067965, -1.296990, -2.624902, -0.790497, 1.570796, 1.638762],accel_mss,speed_ms,0,blend_radius_m)
    |   movel([0.068177, -1.297285, -2.624727, -0.790376, 1.570796, 1.638973],accel_mss,speed_ms,0,blend_radius_m)
    |   movel([0.068448, -1.297463, -2.624622, -0.790304, 1.570796, 1.639244],accel_mss,speed_ms,0,blend_radius_m)
    |   movel([0.068582, -1.297195, -2.624781, -0.790413, 1.570796, 1.639379],accel_mss,speed_ms,0,blend_radius_m)
    |   movel([0.068570, -1.296945, -2.624929, -0.790515, 1.570796, 1.639366],accel_mss,speed_ms,0,blend_radius_m)
    |   movel([0.068283, -1.297098, -2.624839, -0.790453, 1.570796, 1.639079],accel_mss,speed_ms,0,blend_radius_m)
    |   movel([0.068322, -1.296834, -2.624995, -0.790560, 1.570796, 1.639119],accel_mss,speed_ms,0,blend_radius_m)
    |   movel([0.068410, -1.296575, -2.625148, -0.790666, 1.570796, 1.639206],accel_mss,speed_ms,0,blend_radius_m)
    |   movel([0.068413, -1.296331, -2.625292, -0.790766, 1.570796, 1.639209],accel_mss,speed_ms,0,blend_radius_m)
    |   movel([0.068610, -1.296024, -2.625474, -0.790891, 1.570796, 1.639406],accel_mss,speed_ms,0,blend_radius_m)
    |   movel([0.068344, -1.296042, -2.625463, -0.790884, 1.570796, 1.639140],accel_mss,speed_ms,0,blend_radius_m)
    |   movel([0.068247, -1.296349, -2.625281, -0.790758, 1.570796, 1.639043],accel_mss,speed_ms,0,blend_radius_m)
    |   movel([0.068015, -1.296285, -2.625319, -0.790785, 1.570796, 1.638811],accel_mss,speed_ms,0,blend_radius_m)
    |   movel([0.068098, -1.295843, -2.625580, -0.790965, 1.570796, 1.638894],accel_mss,speed_ms,0,blend_radius_m)
    |   movel([0.068346, -1.295534, -2.625763, -0.791092, 1.570796, 1.639142],accel_mss,speed_ms,0,blend_radius_m)
    |   movel([0.068703, -1.295215, -2.625951, -0.791223, 1.570796, 1.639499],accel_mss,speed_ms,0,blend_radius_m)
    |   movel([0.069005, -1.294904, -2.626135, -0.791351, 1.570796, 1.639802],accel_mss,speed_ms,0,blend_radius_m)
    |   movel([0.068736, -1.294446, -2.626405, -0.791539, 1.570796, 1.639533],accel_mss,speed_ms,0,blend_radius_m)
    |   movel([0.068447, -1.294179, -2.626561, -0.791649, 1.570796, 1.639243],accel_mss,speed_ms,0,blend_radius_m)
    |   movel([0.068186, -1.293987, -2.626674, -0.791727, 1.570796, 1.638982],accel_mss,speed_ms,0,blend_radius_m)
    |   movel([0.068055, -1.293698, -2.626844, -0.791847, 1.570796, 1.638851],accel_mss,speed_ms,0,blend_radius_m)
    |   movel([0.068400, -1.293396, -2.627022, -0.791971, 1.570796, 1.639196],accel_mss,speed_ms,0,blend_radius_m)
    |   movel([0.068673, -1.293222, -2.627124, -0.792043, 1.570796, 1.639470],accel_mss,speed_ms,0,blend_radius_m)
    |   movel([0.068591, -1.292993, -2.627259, -0.792138, 1.570796, 1.639387],accel_mss,speed_ms,0,blend_radius_m)
    |   movel([0.068494, -1.292776, -2.627386, -0.792227, 1.570796, 1.639291],accel_mss,speed_ms,0,blend_radius_m)
    |   movel([0.068508, -1.292532, -2.627529, -0.792328, 1.570796, 1.639305],accel_mss,speed_ms,0,blend_radius_m)
    |   movel([0.068313, -1.292435, -2.627586, -0.792368, 1.570796, 1.639109],accel_mss,speed_ms,0,blend_radius_m)
    |   movel([0.068432, -1.292054, -2.627809, -0.792526, 1.570796, 1.639228],accel_mss,speed_ms,0,blend_radius_m)
    |   movel([0.068734, -1.291591, -2.628080, -0.792718, 1.570796, 1.639530],accel_mss,speed_ms,0,blend_radius_m)
    |   movel([0.069080, -1.291360, -2.628215, -0.792814, 1.570796, 1.639876],accel_mss,speed_ms,0,blend_radius_m)
    |   movel([0.069351, -1.291183, -2.628319, -0.792887, 1.570796, 1.640148],accel_mss,speed_ms,0,blend_radius_m)
    |   movel([0.069675, -1.290933, -2.628465, -0.792991, 1.570796, 1.640471],accel_mss,speed_ms,0,blend_radius_m)
    |   movel([0.069973, -1.290833, -2.628523, -0.793033, 1.570796, 1.640769],accel_mss,speed_ms,0,blend_radius_m)
    |   movel([0.070329, -1.290548, -2.628690, -0.793151, 1.570796, 1.641125],accel_mss,speed_ms,0,blend_radius_m)
    |   movel([0.070734, -1.290402, -2.628775, -0.793212, 1.570796, 1.641530],accel_mss,speed_ms,0,blend_radius_m)
    |   movel([0.070848, -1.290597, -2.628661, -0.793131, 1.570796, 1.641644],accel_mss,speed_ms,0,blend_radius_m)
    |   movel([0.070586, -1.290557, -2.628684, -0.793148, 1.570796, 1.641382],accel_mss,speed_ms,0,blend_radius_m)
    |   movel([0.070545, -1.290828, -2.628526, -0.793035, 1.570796, 1.641341],accel_mss,speed_ms,0,blend_radius_m)
    |   movel([0.070287, -1.290805, -2.628540, -0.793044, 1.570796, 1.641083],accel_mss,speed_ms,0,blend_radius_m)
    |   movel([0.070092, -1.291071, -2.628384, -0.792934, 1.570796, 1.640888],accel_mss,speed_ms,0,blend_radius_m)
    |   movel([0.069788, -1.291216, -2.628299, -0.792873, 1.570796, 1.640584],accel_mss,speed_ms,0,blend_radius_m)
    |   movel([0.070023, -1.291249, -2.628280, -0.792860, 1.570796, 1.640820],accel_mss,speed_ms,0,blend_radius_m)
    |   movel([0.070448, -1.291024, -2.628412, -0.792954, 1.570796, 1.641244],accel_mss,speed_ms,0,blend_radius_m)
    |   movel([0.070733, -1.290883, -2.628494, -0.793012, 1.570796, 1.641529],accel_mss,speed_ms,0,blend_radius_m)
    |   movel([0.071014, -1.290753, -2.628570, -0.793066, 1.570796, 1.641811],accel_mss,speed_ms,0,blend_radius_m)
    |   movel([0.071419, -1.290544, -2.628692, -0.793153, 1.570796, 1.642215],accel_mss,speed_ms,0,blend_radius_m)
    |   movel([0.071699, -1.290195, -2.628896, -0.793298, 1.570796, 1.642496],accel_mss,speed_ms,0,blend_radius_m)
    |   movel([0.071397, -1.290344, -2.628808, -0.793236, 1.570796, 1.642193],accel_mss,speed_ms,0,blend_radius_m)
    |   movel([0.071394, -1.290015, -2.629001, -0.793373, 1.570796, 1.642190],accel_mss,speed_ms,0,blend_radius_m)
    |   movel([0.071674, -1.289807, -2.629122, -0.793460, 1.570796, 1.642471],accel_mss,speed_ms,0,blend_radius_m)
    |   movel([0.072099, -1.289622, -2.629230, -0.793537, 1.570796, 1.642895],accel_mss,speed_ms,0,blend_radius_m)
    |   movel([0.072618, -1.289439, -2.629336, -0.793614, 1.570796, 1.643415],accel_mss,speed_ms,0,blend_radius_m)
    |   movel([0.072298, -1.289775, -2.629140, -0.793473, 1.570796, 1.643094],accel_mss,speed_ms,0,blend_radius_m)
    |   movel([0.072072, -1.290052, -2.628979, -0.793358, 1.570796, 1.642868],accel_mss,speed_ms,0,blend_radius_m)
    |   movel([0.072318, -1.290082, -2.628962, -0.793345, 1.570796, 1.643115],accel_mss,speed_ms,0,blend_radius_m)
    |   movel([0.072810, -1.289907, -2.629064, -0.793418, 1.570796, 1.643606],accel_mss,speed_ms,0,blend_radius_m)
    |   movel([0.073098, -1.289924, -2.629053, -0.793411, 1.570796, 1.643895],accel_mss,speed_ms,0,blend_radius_m)
    |   movel([0.073371, -1.289879, -2.629080, -0.793430, 1.570796, 1.644167],accel_mss,speed_ms,0,blend_radius_m)
    |   movel([0.073643, -1.289667, -2.629204, -0.793519, 1.570796, 1.644439],accel_mss,speed_ms,0,blend_radius_m)
    |   movel([0.073422, -1.289556, -2.629268, -0.793565, 1.570796, 1.644218],accel_mss,speed_ms,0,blend_radius_m)
    |   movel([0.073605, -1.289116, -2.629525, -0.793749, 1.570796, 1.644402],accel_mss,speed_ms,0,blend_radius_m)
    |   movel([0.074088, -1.288858, -2.629674, -0.793857, 1.570796, 1.644884],accel_mss,speed_ms,0,blend_radius_m)
    |   movel([0.074586, -1.288774, -2.629723, -0.793892, 1.570796, 1.645382],accel_mss,speed_ms,0,blend_radius_m)
    |   movel([0.075419, -1.288701, -2.629765, -0.793922, 1.570796, 1.646216],accel_mss,speed_ms,0,blend_radius_m)
    |   movel([0.075774, -1.288673, -2.629782, -0.793934, 1.570796, 1.646570],accel_mss,speed_ms,0,blend_radius_m)
    |   movel([0.076162, -1.288635, -2.629804, -0.793950, 1.570796, 1.646959],accel_mss,speed_ms,0,blend_radius_m)
    |   movel([0.076529, -1.288597, -2.629826, -0.793966, 1.570796, 1.647325],accel_mss,speed_ms,0,blend_radius_m)
    |   movel([0.076800, -1.288565, -2.629845, -0.793979, 1.570796, 1.647596],accel_mss,speed_ms,0,blend_radius_m)
    |   movel([0.077294, -1.288560, -2.629848, -0.793981, 1.570796, 1.648090],accel_mss,speed_ms,0,blend_radius_m)
    |   movel([0.077690, -1.288646, -2.629798, -0.793945, 1.570796, 1.648486],accel_mss,speed_ms,0,blend_radius_m)
    |   movel([0.078122, -1.288841, -2.629684, -0.793864, 1.570796, 1.648918],accel_mss,speed_ms,0,blend_radius_m)
    |   movel([0.078432, -1.288951, -2.629621, -0.793818, 1.570796, 1.649228],accel_mss,speed_ms,0,blend_radius_m)
    |   movel([0.078708, -1.289007, -2.629588, -0.793794, 1.570796, 1.649504],accel_mss,speed_ms,0,blend_radius_m)
    |   movel([0.079022, -1.289032, -2.629573, -0.793784, 1.570796, 1.649819],accel_mss,speed_ms,0,blend_radius_m)
    |   movel([0.079477, -1.289125, -2.629519, -0.793745, 1.570796, 1.650273],accel_mss,speed_ms,0,blend_radius_m)
    |   movel([0.080017, -1.289405, -2.629356, -0.793628, 1.570796, 1.650813],accel_mss,speed_ms,0,blend_radius_m)
    |   movel([0.080490, -1.289761, -2.629149, -0.793479, 1.570796, 1.651286],accel_mss,speed_ms,0,blend_radius_m)
    |   movel([0.080723, -1.290104, -2.628949, -0.793336, 1.570796, 1.651519],accel_mss,speed_ms,0,blend_radius_m)
    |   movel([0.080790, -1.290461, -2.628740, -0.793187, 1.570796, 1.651586],accel_mss,speed_ms,0,blend_radius_m)
    |   movel([0.080755, -1.290906, -2.628480, -0.793002, 1.570796, 1.651551],accel_mss,speed_ms,0,blend_radius_m)
    |   movel([0.080623, -1.291367, -2.628211, -0.792811, 1.570796, 1.651420],accel_mss,speed_ms,0,blend_radius_m)
    |   movel([0.080414, -1.291769, -2.627976, -0.792644, 1.570796, 1.651210],accel_mss,speed_ms,0,blend_radius_m)
    |   movel([0.080193, -1.292059, -2.627806, -0.792524, 1.570796, 1.650990],accel_mss,speed_ms,0,blend_radius_m)
    |   movel([0.079916, -1.292349, -2.627636, -0.792404, 1.570796, 1.650712],accel_mss,speed_ms,0,blend_radius_m)
    |   movel([0.079600, -1.292623, -2.627475, -0.792290, 1.570796, 1.650396],accel_mss,speed_ms,0,blend_radius_m)
    |   movel([0.079260, -1.292868, -2.627332, -0.792189, 1.570796, 1.650056],accel_mss,speed_ms,0,blend_radius_m)
    |   movel([0.079132, -1.292699, -2.627431, -0.792259, 1.570796, 1.649929],accel_mss,speed_ms,0,blend_radius_m)
    |   movel([0.078790, -1.293064, -2.627217, -0.792108, 1.570796, 1.649586],accel_mss,speed_ms,0,blend_radius_m)
    |   movel([0.078548, -1.293294, -2.627082, -0.792013, 1.570796, 1.649345],accel_mss,speed_ms,0,blend_radius_m)
    |   movel([0.078210, -1.293734, -2.626823, -0.791832, 1.570796, 1.649006],accel_mss,speed_ms,0,blend_radius_m)
    |   movel([0.078166, -1.294015, -2.626658, -0.791716, 1.570796, 1.648962],accel_mss,speed_ms,0,blend_radius_m)
    |   movel([0.078357, -1.294349, -2.626462, -0.791579, 1.570796, 1.649153],accel_mss,speed_ms,0,blend_radius_m)
    |   movel([0.078391, -1.294602, -2.626313, -0.791475, 1.570796, 1.649187],accel_mss,speed_ms,0,blend_radius_m)
    |   movel([0.078328, -1.294883, -2.626147, -0.791359, 1.570796, 1.649124],accel_mss,speed_ms,0,blend_radius_m)
    |   movel([0.078048, -1.295310, -2.625895, -0.791184, 1.570796, 1.648844],accel_mss,speed_ms,0,blend_radius_m)
    |   movel([0.078070, -1.295548, -2.625754, -0.791086, 1.570796, 1.648866],accel_mss,speed_ms,0,blend_radius_m)
    |   movel([0.077797, -1.295930, -2.625529, -0.790930, 1.570796, 1.648593],accel_mss,speed_ms,0,blend_radius_m)
    |   movel([0.077543, -1.296213, -2.625362, -0.790814, 1.570796, 1.648340],accel_mss,speed_ms,0,blend_radius_m)
    |   movel([0.077141, -1.296453, -2.625220, -0.790716, 1.570796, 1.647937],accel_mss,speed_ms,0,blend_radius_m)
    |   movel([0.076881, -1.296662, -2.625096, -0.790630, 1.570796, 1.647677],accel_mss,speed_ms,0,blend_radius_m)
    |   movel([0.076380, -1.296832, -2.624996, -0.790561, 1.570796, 1.647176],accel_mss,speed_ms,0,blend_radius_m)
    |   movel([0.076038, -1.297953, -2.624332, -0.790105, 1.570796, 1.646834],accel_mss,speed_ms,0,blend_radius_m)
    |   movel([0.075953, -1.298382, -2.624077, -0.789930, 1.570796, 1.646749],accel_mss,speed_ms,0,blend_radius_m)
    |   movel([0.075814, -1.298681, -2.623899, -0.789809, 1.570796, 1.646610],accel_mss,speed_ms,0,blend_radius_m)
    |   movel([0.075570, -1.298998, -2.623711, -0.789680, 1.570796, 1.646366],accel_mss,speed_ms,0,blend_radius_m)
    |   movel([0.075189, -1.299340, -2.623508, -0.789542, 1.570796, 1.645986],accel_mss,speed_ms,0,blend_radius_m)
    |   movel([0.074854, -1.299474, -2.623428, -0.789487, 1.570796, 1.645650],accel_mss,speed_ms,0,blend_radius_m)
    |   movel([0.074612, -1.299705, -2.623290, -0.789394, 1.570796, 1.645408],accel_mss,speed_ms,0,blend_radius_m)
    |   movel([0.074370, -1.299617, -2.623343, -0.789430, 1.570796, 1.645166],accel_mss,speed_ms,0,blend_radius_m)
    |   movel([0.074338, -1.299900, -2.623174, -0.789315, 1.570796, 1.645134],accel_mss,speed_ms,0,blend_radius_m)
    |   movel([0.073982, -1.300051, -2.623084, -0.789254, 1.570796, 1.644779],accel_mss,speed_ms,0,blend_radius_m)
    |   speed_ms = 0.003
    |   movel([0.073982, -1.303545, -2.624704, -0.784140, 1.570796, 1.644779],accel_mss,speed_ms,0,blend_radius_m)
    |   speed_ms = 0.007
    |   movel([0.073932, -1.303284, -2.624861, -0.784245, 1.570796, 1.644728],accel_mss,speed_ms,0,blend_radius_m)
    |   movel([0.074261, -1.303044, -2.625004, -0.784341, 1.570796, 1.645057],accel_mss,speed_ms,0,blend_radius_m)
    |   movel([0.074673, -1.302820, -2.625138, -0.784431, 1.570796, 1.645470],accel_mss,speed_ms,0,blend_radius_m)
    |   movel([0.074331, -1.302852, -2.625119, -0.784418, 1.570796, 1.645127],accel_mss,speed_ms,0,blend_radius_m)
    |   movel([0.073782, -1.303089, -2.624977, -0.784323, 1.570796, 1.644579],accel_mss,speed_ms,0,blend_radius_m)
    |   movel([0.072985, -1.303366, -2.624811, -0.784211, 1.570796, 1.643781],accel_mss,speed_ms,0,blend_radius_m)
    |   movel([0.072179, -1.303619, -2.624660, -0.784110, 1.570796, 1.642975],accel_mss,speed_ms,0,blend_radius_m)
    |   movel([0.071902, -1.303597, -2.624673, -0.784119, 1.570796, 1.642698],accel_mss,speed_ms,0,blend_radius_m)
    |   movel([0.071682, -1.303891, -2.624497, -0.784001, 1.570796, 1.642478],accel_mss,speed_ms,0,blend_radius_m)
    |   movel([0.071302, -1.304085, -2.624380, -0.783923, 1.570796, 1.642098],accel_mss,speed_ms,0,blend_radius_m)
    |   movel([0.071480, -1.303802, -2.624551, -0.784037, 1.570796, 1.642277],accel_mss,speed_ms,0,blend_radius_m)
    |   movel([0.071194, -1.303858, -2.624517, -0.784014, 1.570796, 1.641991],accel_mss,speed_ms,0,blend_radius_m)
    |   movel([0.070917, -1.304036, -2.624410, -0.783943, 1.570796, 1.641714],accel_mss,speed_ms,0,blend_radius_m)
    |   movel([0.070724, -1.303876, -2.624506, -0.784007, 1.570796, 1.641520],accel_mss,speed_ms,0,blend_radius_m)
    |   movel([0.070555, -1.303705, -2.624608, -0.784075, 1.570796, 1.641352],accel_mss,speed_ms,0,blend_radius_m)
    |   movel([0.070266, -1.303698, -2.624613, -0.784078, 1.570796, 1.641063],accel_mss,speed_ms,0,blend_radius_m)
    |   movel([0.070498, -1.303789, -2.624558, -0.784042, 1.570796, 1.641294],accel_mss,speed_ms,0,blend_radius_m)
    |   movel([0.070207, -1.303999, -2.624432, -0.783958, 1.570796, 1.641004],accel_mss,speed_ms,0,blend_radius_m)
    |   movel([0.069999, -1.303927, -2.624476, -0.783987, 1.570796, 1.640795],accel_mss,speed_ms,0,blend_radius_m)
    |   movel([0.069864, -1.303770, -2.624569, -0.784049, 1.570796, 1.640660],accel_mss,speed_ms,0,blend_radius_m)
    |   movel([0.069616, -1.303985, -2.624441, -0.783964, 1.570796, 1.640412],accel_mss,speed_ms,0,blend_radius_m)
    |   movel([0.069394, -1.303915, -2.624483, -0.783992, 1.570796, 1.640190],accel_mss,speed_ms,0,blend_radius_m)
